(* Logix 5000 project; controller QW361 vendor 1 type 14 code 107 rev 32.11; software revision 32.00; part 12 of 20 *)

        [1618].time.Day := 29, [1618].time.Hour := 12, [1618].time.Minute := 24, [1618].time.Second := 59, [1618].time.DST_ON := 1, [1619].log_data[0].min := 1.0, [1619].log_data[0].max := 1.0, [1619].log_data[0].total := 300.0, [1619].log_data[0].time := 300.0, [1619].log_data[0].minminute := 25, [1619].log_data[0].maxminute := 25, [1619].log_data[0].valid := 1, [1619].log_data[1].valid := 1, [1619].log_data[2].valid := 1, [1619].log_data[3].valid := 1, [1619].log_data[4].valid := 1, [1619].time.Year := 2022, [1619].time.Month := 4, [1619].time.Day := 29, [1619].time.Hour := 12, [1619].time.Minute := 29, [1619].time.Second := 59, [1619].time.DST_ON := 1, [1620].log_data[0].min := 1.0, [1620].log_data[0].max := 1.0, [1620].log_data[0].total := 300.0, [1620].log_data[0].time := 300.0, [1620].log_data[0].minminute := 30, [1620].log_data[0].maxminute := 30, [1620].log_data[0].valid := 1, [1620].log_data[1].valid := 1, [1620].log_data[2].valid := 1, [1620].log_data[3].valid := 1, [1620].log_data[4].valid := 1, [1620].time.Year := 2022, [1620].time.Month := 4, [1620].time.Day := 29, [1620].time.Hour := 12, [1620].time.Minute := 34, [1620].time.Second := 59, [1620].time.DST_ON := 1, [1621].log_data[0].min := 1.0, [1621].log_data[0].max := 1.0, [1621].log_data[0].total := 300.0, [1621].log_data[0].time := 300.0, [1621].log_data[0].minminute := 35, [1621].log_data[0].maxminute := 35, [1621].log_data[0].valid := 1, [1621].log_data[1].valid := 1, [1621].log_data[2].valid := 1, [1621].log_data[3].valid := 1, [1621].log_data[4].valid := 1, [1621].time.Year := 2022, [1621].time.Month := 4, [1621].time.Day := 29, [1621].time.Hour := 12, [1621].time.Minute := 39, [1621].time.Second := 59, [1621].time.DST_ON := 1, [1622].log_data[0].min := 1.0,
        [1622].log_data[0].max := 1.0, [1622].log_data[0].total := 300.0, [1622].log_data[0].time := 300.0, [1622].log_data[0].minminute := 40, [1622].log_data[0].maxminute := 40, [1622].log_data[0].valid := 1, [1622].log_data[1].valid := 1, [1622].log_data[2].valid := 1, [1622].log_data[3].valid := 1, [1622].log_data[4].valid := 1, [1622].time.Year := 2022, [1622].time.Month := 4, [1622].time.Day := 29, [1622].time.Hour := 12, [1622].time.Minute := 44, [1622].time.Second := 59, [1622].time.DST_ON := 1, [1623].log_data[0].min := 1.0, [1623].log_data[0].max := 1.0, [1623].log_data[0].total := 300.0, [1623].log_data[0].time := 300.0, [1623].log_data[0].minminute := 45, [1623].log_data[0].maxminute := 45, [1623].log_data[0].valid := 1, [1623].log_data[1].valid := 1, [1623].log_data[2].valid := 1, [1623].log_data[3].valid := 1, [1623].log_data[4].valid := 1, [1623].time.Year := 2022, [1623].time.Month := 4, [1623].time.Day := 29, [1623].time.Hour := 12, [1623].time.Minute := 49, [1623].time.Second := 59, [1623].time.DST_ON := 1, [1624].log_data[0].min := 1.0, [1624].log_data[0].max := 1.0, [1624].log_data[0].total := 300.0, [1624].log_data[0].time := 300.0, [1624].log_data[0].minminute := 50, [1624].log_data[0].maxminute := 50, [1624].log_data[0].valid := 1, [1624].log_data[1].valid := 1, [1624].log_data[2].valid := 1, [1624].log_data[3].valid := 1, [1624].log_data[4].valid := 1, [1624].time.Year := 2022, [1624].time.Month := 4, [1624].time.Day := 29, [1624].time.Hour := 12, [1624].time.Minute := 54, [1624].time.Second := 59, [1624].time.DST_ON := 1, [1625].log_data[0].min := 1.0, [1625].log_data[0].max := 1.0, [1625].log_data[0].total := 300.0, [1625].log_data[0].time := 300.0, [1625].log_data[0].minminute := 55, [1625].log_data[0].maxminute := 55, [1625].log_data[0].valid := 1,
        [1625].log_data[1].valid := 1, [1625].log_data[2].valid := 1, [1625].log_data[3].valid := 1, [1625].log_data[4].valid := 1, [1625].time.Year := 2022, [1625].time.Month := 4, [1625].time.Day := 29, [1625].time.Hour := 12, [1625].time.Minute := 59, [1625].time.Second := 59, [1625].time.DST_ON := 1, [1626].log_data[0].min := 1.0, [1626].log_data[0].max := 1.0, [1626].log_data[0].total := 300.0, [1626].log_data[0].time := 300.0, [1626].log_data[0].valid := 1, [1626].log_data[1].valid := 1, [1626].log_data[2].valid := 1, [1626].log_data[3].valid := 1, [1626].log_data[4].valid := 1, [1626].time.Year := 2022, [1626].time.Month := 4, [1626].time.Day := 29, [1626].time.Hour := 13, [1626].time.Minute := 4, [1626].time.Second := 59, [1626].time.DST_ON := 1, [1627].log_data[0].min := 1.0, [1627].log_data[0].max := 1.0, [1627].log_data[0].total := 300.0, [1627].log_data[0].time := 300.0, [1627].log_data[0].minminute := 5, [1627].log_data[0].maxminute := 5, [1627].log_data[0].valid := 1, [1627].log_data[1].valid := 1, [1627].log_data[2].valid := 1, [1627].log_data[3].valid := 1, [1627].log_data[4].valid := 1, [1627].time.Year := 2022, [1627].time.Month := 4, [1627].time.Day := 29, [1627].time.Hour := 13, [1627].time.Minute := 9, [1627].time.Second := 59, [1627].time.DST_ON := 1, [1628].log_data[0].min := 1.0, [1628].log_data[0].max := 1.0, [1628].log_data[0].total := 300.0, [1628].log_data[0].time := 300.0, [1628].log_data[0].minminute := 10, [1628].log_data[0].maxminute := 10, [1628].log_data[0].valid := 1, [1628].log_data[1].valid := 1, [1628].log_data[2].valid := 1, [1628].log_data[3].valid := 1, [1628].log_data[4].valid := 1, [1628].time.Year := 2022, [1628].time.Month := 4, [1628].time.Day := 29, [1628].time.Hour := 13,
        [1628].time.Minute := 14, [1628].time.Second := 59, [1628].time.DST_ON := 1, [1629].log_data[0].min := 1.0, [1629].log_data[0].max := 1.0, [1629].log_data[0].total := 300.0, [1629].log_data[0].time := 300.0, [1629].log_data[0].minminute := 15, [1629].log_data[0].maxminute := 15, [1629].log_data[0].valid := 1, [1629].log_data[1].valid := 1, [1629].log_data[2].valid := 1, [1629].log_data[3].valid := 1, [1629].log_data[4].valid := 1, [1629].time.Year := 2022, [1629].time.Month := 4, [1629].time.Day := 29, [1629].time.Hour := 13, [1629].time.Minute := 19, [1629].time.Second := 59, [1629].time.DST_ON := 1, [1630].log_data[0].min := 1.0, [1630].log_data[0].max := 1.0, [1630].log_data[0].total := 300.0, [1630].log_data[0].time := 300.0, [1630].log_data[0].minminute := 20, [1630].log_data[0].maxminute := 20, [1630].log_data[0].valid := 1, [1630].log_data[1].valid := 1, [1630].log_data[2].valid := 1, [1630].log_data[3].valid := 1, [1630].log_data[4].valid := 1, [1630].time.Year := 2022, [1630].time.Month := 4, [1630].time.Day := 29, [1630].time.Hour := 13, [1630].time.Minute := 24, [1630].time.Second := 59, [1630].time.DST_ON := 1, [1631].log_data[0].min := 1.0, [1631].log_data[0].max := 1.0, [1631].log_data[0].total := 300.0, [1631].log_data[0].time := 300.0, [1631].log_data[0].minminute := 25, [1631].log_data[0].maxminute := 25, [1631].log_data[0].valid := 1, [1631].log_data[1].valid := 1, [1631].log_data[2].valid := 1, [1631].log_data[3].valid := 1, [1631].log_data[4].valid := 1, [1631].time.Year := 2022, [1631].time.Month := 4, [1631].time.Day := 29, [1631].time.Hour := 13, [1631].time.Minute := 29, [1631].time.Second := 59, [1631].time.DST_ON := 1, [1632].log_data[0].min := 1.0, [1632].log_data[0].max := 1.0, [1632].log_data[0].total := 300.0,
        [1632].log_data[0].time := 300.0, [1632].log_data[0].minminute := 30, [1632].log_data[0].maxminute := 30, [1632].log_data[0].valid := 1, [1632].log_data[1].valid := 1, [1632].log_data[2].valid := 1, [1632].log_data[3].valid := 1, [1632].log_data[4].valid := 1, [1632].time.Year := 2022, [1632].time.Month := 4, [1632].time.Day := 29, [1632].time.Hour := 13, [1632].time.Minute := 34, [1632].time.Second := 59, [1632].time.DST_ON := 1, [1633].log_data[0].min := 1.0, [1633].log_data[0].max := 1.0, [1633].log_data[0].total := 300.001, [1633].log_data[0].time := 300.001, [1633].log_data[0].minminute := 35, [1633].log_data[0].maxminute := 35, [1633].log_data[0].valid := 1, [1633].log_data[1].valid := 1, [1633].log_data[2].valid := 1, [1633].log_data[3].valid := 1, [1633].log_data[4].valid := 1, [1633].time.Year := 2022, [1633].time.Month := 4, [1633].time.Day := 29, [1633].time.Hour := 13, [1633].time.Minute := 39, [1633].time.Second := 59, [1633].time.DST_ON := 1, [1634].log_data[0].min := 1.0, [1634].log_data[0].max := 1.0, [1634].log_data[0].total := 300.0, [1634].log_data[0].time := 300.0, [1634].log_data[0].minminute := 40, [1634].log_data[0].maxminute := 40, [1634].log_data[0].valid := 1, [1634].log_data[1].valid := 1, [1634].log_data[2].valid := 1, [1634].log_data[3].valid := 1, [1634].log_data[4].valid := 1, [1634].time.Year := 2022, [1634].time.Month := 4, [1634].time.Day := 29, [1634].time.Hour := 13, [1634].time.Minute := 44, [1634].time.Second := 59, [1634].time.DST_ON := 1, [1635].log_data[0].min := 1.0, [1635].log_data[0].max := 1.0, [1635].log_data[0].total := 300.0, [1635].log_data[0].time := 300.0, [1635].log_data[0].minminute := 45, [1635].log_data[0].maxminute := 45, [1635].log_data[0].valid := 1, [1635].log_data[1].valid := 1, [1635].log_data[2].valid := 1,
        [1635].log_data[3].valid := 1, [1635].log_data[4].valid := 1, [1635].time.Year := 2022, [1635].time.Month := 4, [1635].time.Day := 29, [1635].time.Hour := 13, [1635].time.Minute := 49, [1635].time.Second := 59, [1635].time.DST_ON := 1, [1636].log_data[0].min := 1.0, [1636].log_data[0].max := 1.0, [1636].log_data[0].total := 300.0, [1636].log_data[0].time := 300.0, [1636].log_data[0].minminute := 50, [1636].log_data[0].maxminute := 50, [1636].log_data[0].valid := 1, [1636].log_data[1].valid := 1, [1636].log_data[2].valid := 1, [1636].log_data[3].valid := 1, [1636].log_data[4].valid := 1, [1636].time.Year := 2022, [1636].time.Month := 4, [1636].time.Day := 29, [1636].time.Hour := 13, [1636].time.Minute := 54, [1636].time.Second := 59, [1636].time.DST_ON := 1, [1637].log_data[0].min := 1.0, [1637].log_data[0].max := 1.0, [1637].log_data[0].total := 300.0, [1637].log_data[0].time := 300.0, [1637].log_data[0].minminute := 55, [1637].log_data[0].maxminute := 55, [1637].log_data[0].valid := 1, [1637].log_data[1].valid := 1, [1637].log_data[2].valid := 1, [1637].log_data[3].valid := 1, [1637].log_data[4].valid := 1, [1637].time.Year := 2022, [1637].time.Month := 4, [1637].time.Day := 29, [1637].time.Hour := 13, [1637].time.Minute := 59, [1637].time.Second := 59, [1637].time.DST_ON := 1, [1638].log_data[0].min := 1.0, [1638].log_data[0].max := 1.0, [1638].log_data[0].total := 300.0, [1638].log_data[0].time := 300.0, [1638].log_data[0].valid := 1, [1638].log_data[1].valid := 1, [1638].log_data[2].valid := 1, [1638].log_data[3].valid := 1, [1638].log_data[4].valid := 1, [1638].time.Year := 2022, [1638].time.Month := 4, [1638].time.Day := 29, [1638].time.Hour := 14, [1638].time.Minute := 4, [1638].time.Second := 59,
        [1638].time.DST_ON := 1, [1639].log_data[0].min := 1.0, [1639].log_data[0].max := 1.0, [1639].log_data[0].total := 300.0, [1639].log_data[0].time := 300.0, [1639].log_data[0].minminute := 5, [1639].log_data[0].maxminute := 5, [1639].log_data[0].valid := 1, [1639].log_data[1].valid := 1, [1639].log_data[2].valid := 1, [1639].log_data[3].valid := 1, [1639].log_data[4].valid := 1, [1639].time.Year := 2022, [1639].time.Month := 4, [1639].time.Day := 29, [1639].time.Hour := 14, [1639].time.Minute := 9, [1639].time.Second := 59, [1639].time.DST_ON := 1, [1640].log_data[0].min := 1.0, [1640].log_data[0].max := 1.0, [1640].log_data[0].total := 300.0, [1640].log_data[0].time := 300.0, [1640].log_data[0].minminute := 10, [1640].log_data[0].maxminute := 10, [1640].log_data[0].valid := 1, [1640].log_data[1].valid := 1, [1640].log_data[2].valid := 1, [1640].log_data[3].valid := 1, [1640].log_data[4].valid := 1, [1640].time.Year := 2022, [1640].time.Month := 4, [1640].time.Day := 29, [1640].time.Hour := 14, [1640].time.Minute := 14, [1640].time.Second := 59, [1640].time.DST_ON := 1, [1641].log_data[0].min := 1.0, [1641].log_data[0].max := 1.0, [1641].log_data[0].total := 299.999, [1641].log_data[0].time := 299.999, [1641].log_data[0].minminute := 15, [1641].log_data[0].maxminute := 15, [1641].log_data[0].valid := 1, [1641].log_data[1].valid := 1, [1641].log_data[2].valid := 1, [1641].log_data[3].valid := 1, [1641].log_data[4].valid := 1, [1641].time.Year := 2022, [1641].time.Month := 4, [1641].time.Day := 29, [1641].time.Hour := 14, [1641].time.Minute := 19, [1641].time.Second := 59, [1641].time.DST_ON := 1, [1642].log_data[0].min := 1.0, [1642].log_data[0].max := 1.0, [1642].log_data[0].total := 300.0, [1642].log_data[0].time := 300.0, [1642].log_data[0].minminute := 20,
        [1642].log_data[0].maxminute := 20, [1642].log_data[0].valid := 1, [1642].log_data[1].valid := 1, [1642].log_data[2].valid := 1, [1642].log_data[3].valid := 1, [1642].log_data[4].valid := 1, [1642].time.Year := 2022, [1642].time.Month := 4, [1642].time.Day := 29, [1642].time.Hour := 14, [1642].time.Minute := 24, [1642].time.Second := 59, [1642].time.DST_ON := 1, [1643].log_data[0].min := 1.0, [1643].log_data[0].max := 1.0, [1643].log_data[0].total := 300.0, [1643].log_data[0].time := 300.0, [1643].log_data[0].minminute := 25, [1643].log_data[0].maxminute := 25, [1643].log_data[0].valid := 1, [1643].log_data[1].valid := 1, [1643].log_data[2].valid := 1, [1643].log_data[3].valid := 1, [1643].log_data[4].valid := 1, [1643].time.Year := 2022, [1643].time.Month := 4, [1643].time.Day := 29, [1643].time.Hour := 14, [1643].time.Minute := 29, [1643].time.Second := 59, [1643].time.DST_ON := 1, [1644].log_data[0].min := 1.0, [1644].log_data[0].max := 1.0, [1644].log_data[0].total := 300.0, [1644].log_data[0].time := 300.0, [1644].log_data[0].minminute := 30, [1644].log_data[0].maxminute := 30, [1644].log_data[0].valid := 1, [1644].log_data[1].valid := 1, [1644].log_data[2].valid := 1, [1644].log_data[3].valid := 1, [1644].log_data[4].valid := 1, [1644].time.Year := 2022, [1644].time.Month := 4, [1644].time.Day := 29, [1644].time.Hour := 14, [1644].time.Minute := 34, [1644].time.Second := 59, [1644].time.DST_ON := 1, [1645].log_data[0].min := 1.0, [1645].log_data[0].max := 1.0, [1645].log_data[0].total := 300.0, [1645].log_data[0].time := 300.0, [1645].log_data[0].minminute := 35, [1645].log_data[0].maxminute := 35, [1645].log_data[0].valid := 1, [1645].log_data[1].valid := 1, [1645].log_data[2].valid := 1, [1645].log_data[3].valid := 1, [1645].log_data[4].valid := 1,
        [1645].time.Year := 2022, [1645].time.Month := 4, [1645].time.Day := 29, [1645].time.Hour := 14, [1645].time.Minute := 39, [1645].time.Second := 59, [1645].time.DST_ON := 1, [1646].log_data[0].min := 1.0, [1646].log_data[0].max := 1.0, [1646].log_data[0].total := 300.0, [1646].log_data[0].time := 300.0, [1646].log_data[0].minminute := 40, [1646].log_data[0].maxminute := 40, [1646].log_data[0].valid := 1, [1646].log_data[1].valid := 1, [1646].log_data[2].valid := 1, [1646].log_data[3].valid := 1, [1646].log_data[4].valid := 1, [1646].time.Year := 2022, [1646].time.Month := 4, [1646].time.Day := 29, [1646].time.Hour := 14, [1646].time.Minute := 44, [1646].time.Second := 59, [1646].time.DST_ON := 1, [1647].log_data[0].min := 1.0, [1647].log_data[0].max := 1.0, [1647].log_data[0].total := 300.0, [1647].log_data[0].time := 300.0, [1647].log_data[0].minminute := 45, [1647].log_data[0].maxminute := 45, [1647].log_data[0].valid := 1, [1647].log_data[1].valid := 1, [1647].log_data[2].valid := 1, [1647].log_data[3].valid := 1, [1647].log_data[4].valid := 1, [1647].time.Year := 2022, [1647].time.Month := 4, [1647].time.Day := 29, [1647].time.Hour := 14, [1647].time.Minute := 49, [1647].time.Second := 59, [1647].time.DST_ON := 1, [1648].log_data[0].min := 1.0, [1648].log_data[0].max := 1.0, [1648].log_data[0].total := 300.0, [1648].log_data[0].time := 300.0, [1648].log_data[0].minminute := 50, [1648].log_data[0].maxminute := 50, [1648].log_data[0].valid := 1, [1648].log_data[1].valid := 1, [1648].log_data[2].valid := 1, [1648].log_data[3].valid := 1, [1648].log_data[4].valid := 1, [1648].time.Year := 2022, [1648].time.Month := 4, [1648].time.Day := 29, [1648].time.Hour := 14, [1648].time.Minute := 54, [1648].time.Second := 59,
        [1648].time.DST_ON := 1, [1649].log_data[0].min := 1.0, [1649].log_data[0].max := 1.0, [1649].log_data[0].total := 300.0, [1649].log_data[0].time := 300.0, [1649].log_data[0].minminute := 55, [1649].log_data[0].maxminute := 55, [1649].log_data[0].valid := 1, [1649].log_data[1].valid := 1, [1649].log_data[2].valid := 1, [1649].log_data[3].valid := 1, [1649].log_data[4].valid := 1, [1649].time.Year := 2022, [1649].time.Month := 4, [1649].time.Day := 29, [1649].time.Hour := 14, [1649].time.Minute := 59, [1649].time.Second := 59, [1649].time.DST_ON := 1, [1650].log_data[0].min := 1.0, [1650].log_data[0].max := 1.0, [1650].log_data[0].total := 300.0, [1650].log_data[0].time := 300.0, [1650].log_data[0].valid := 1, [1650].log_data[1].valid := 1, [1650].log_data[2].valid := 1, [1650].log_data[3].valid := 1, [1650].log_data[4].valid := 1, [1650].time.Year := 2022, [1650].time.Month := 4, [1650].time.Day := 29, [1650].time.Hour := 15, [1650].time.Minute := 4, [1650].time.Second := 59, [1650].time.DST_ON := 1, [1651].log_data[0].min := 1.0, [1651].log_data[0].max := 1.0, [1651].log_data[0].total := 300.0, [1651].log_data[0].time := 300.0, [1651].log_data[0].minminute := 5, [1651].log_data[0].maxminute := 5, [1651].log_data[0].valid := 1, [1651].log_data[1].valid := 1, [1651].log_data[2].valid := 1, [1651].log_data[3].valid := 1, [1651].log_data[4].valid := 1, [1651].time.Year := 2022, [1651].time.Month := 4, [1651].time.Day := 29, [1651].time.Hour := 15, [1651].time.Minute := 9, [1651].time.Second := 59, [1651].time.DST_ON := 1, [1652].log_data[0].min := 1.0, [1652].log_data[0].max := 1.0, [1652].log_data[0].total := 300.0, [1652].log_data[0].time := 300.0, [1652].log_data[0].minminute := 10, [1652].log_data[0].maxminute := 10, [1652].log_data[0].valid := 1,
        [1652].log_data[1].valid := 1, [1652].log_data[2].valid := 1, [1652].log_data[3].valid := 1, [1652].log_data[4].valid := 1, [1652].time.Year := 2022, [1652].time.Month := 4, [1652].time.Day := 29, [1652].time.Hour := 15, [1652].time.Minute := 14, [1652].time.Second := 59, [1652].time.DST_ON := 1, [1653].log_data[0].min := 1.0, [1653].log_data[0].max := 1.0, [1653].log_data[0].total := 300.0, [1653].log_data[0].time := 300.0, [1653].log_data[0].minminute := 15, [1653].log_data[0].maxminute := 15, [1653].log_data[0].valid := 1, [1653].log_data[1].valid := 1, [1653].log_data[2].valid := 1, [1653].log_data[3].valid := 1, [1653].log_data[4].valid := 1, [1653].time.Year := 2022, [1653].time.Month := 4, [1653].time.Day := 29, [1653].time.Hour := 15, [1653].time.Minute := 19, [1653].time.Second := 59, [1653].time.DST_ON := 1, [1654].log_data[0].min := 1.0, [1654].log_data[0].max := 1.0, [1654].log_data[0].total := 300.0, [1654].log_data[0].time := 300.0, [1654].log_data[0].minminute := 20, [1654].log_data[0].maxminute := 20, [1654].log_data[0].valid := 1, [1654].log_data[1].valid := 1, [1654].log_data[2].valid := 1, [1654].log_data[3].valid := 1, [1654].log_data[4].valid := 1, [1654].time.Year := 2022, [1654].time.Month := 4, [1654].time.Day := 29, [1654].time.Hour := 15, [1654].time.Minute := 24, [1654].time.Second := 59, [1654].time.DST_ON := 1, [1655].log_data[0].min := 1.0, [1655].log_data[0].max := 1.0, [1655].log_data[0].total := 300.0, [1655].log_data[0].time := 300.0, [1655].log_data[0].minminute := 25, [1655].log_data[0].maxminute := 25, [1655].log_data[0].valid := 1, [1655].log_data[1].valid := 1, [1655].log_data[2].valid := 1, [1655].log_data[3].valid := 1, [1655].log_data[4].valid := 1, [1655].time.Year := 2022, [1655].time.Month := 4,
        [1655].time.Day := 29, [1655].time.Hour := 15, [1655].time.Minute := 29, [1655].time.Second := 59, [1655].time.DST_ON := 1, [1656].log_data[0].min := 1.0, [1656].log_data[0].max := 1.0, [1656].log_data[0].total := 300.001, [1656].log_data[0].time := 300.001, [1656].log_data[0].minminute := 30, [1656].log_data[0].maxminute := 30, [1656].log_data[0].valid := 1, [1656].log_data[1].valid := 1, [1656].log_data[2].valid := 1, [1656].log_data[3].valid := 1, [1656].log_data[4].valid := 1, [1656].time.Year := 2022, [1656].time.Month := 4, [1656].time.Day := 29, [1656].time.Hour := 15, [1656].time.Minute := 34, [1656].time.Second := 59, [1656].time.DST_ON := 1, [1657].log_data[0].min := 1.0, [1657].log_data[0].max := 1.0, [1657].log_data[0].total := 300.0, [1657].log_data[0].time := 300.0, [1657].log_data[0].minminute := 35, [1657].log_data[0].maxminute := 35, [1657].log_data[0].valid := 1, [1657].log_data[1].valid := 1, [1657].log_data[2].valid := 1, [1657].log_data[3].valid := 1, [1657].log_data[4].valid := 1, [1657].time.Year := 2022, [1657].time.Month := 4, [1657].time.Day := 29, [1657].time.Hour := 15, [1657].time.Minute := 39, [1657].time.Second := 59, [1657].time.DST_ON := 1, [1658].log_data[0].min := 1.0, [1658].log_data[0].max := 1.0, [1658].log_data[0].total := 300.0, [1658].log_data[0].time := 300.0, [1658].log_data[0].minminute := 40, [1658].log_data[0].maxminute := 40, [1658].log_data[0].valid := 1, [1658].log_data[1].valid := 1, [1658].log_data[2].valid := 1, [1658].log_data[3].valid := 1, [1658].log_data[4].valid := 1, [1658].time.Year := 2022, [1658].time.Month := 4, [1658].time.Day := 29, [1658].time.Hour := 15, [1658].time.Minute := 44, [1658].time.Second := 59, [1658].time.DST_ON := 1, [1659].log_data[0].min := 1.0,
        [1659].log_data[0].max := 1.0, [1659].log_data[0].total := 300.0, [1659].log_data[0].time := 300.0, [1659].log_data[0].minminute := 45, [1659].log_data[0].maxminute := 45, [1659].log_data[0].valid := 1, [1659].log_data[1].valid := 1, [1659].log_data[2].valid := 1, [1659].log_data[3].valid := 1, [1659].log_data[4].valid := 1, [1659].time.Year := 2022, [1659].time.Month := 4, [1659].time.Day := 29, [1659].time.Hour := 15, [1659].time.Minute := 49, [1659].time.Second := 59, [1659].time.DST_ON := 1, [1660].log_data[0].min := 1.0, [1660].log_data[0].max := 1.0, [1660].log_data[0].total := 300.0, [1660].log_data[0].time := 300.0, [1660].log_data[0].minminute := 50, [1660].log_data[0].maxminute := 50, [1660].log_data[0].valid := 1, [1660].log_data[1].valid := 1, [1660].log_data[2].valid := 1, [1660].log_data[3].valid := 1, [1660].log_data[4].valid := 1, [1660].time.Year := 2022, [1660].time.Month := 4, [1660].time.Day := 29, [1660].time.Hour := 15, [1660].time.Minute := 54, [1660].time.Second := 59, [1660].time.DST_ON := 1, [1661].log_data[0].min := 1.0, [1661].log_data[0].max := 1.0, [1661].log_data[0].total := 300.0, [1661].log_data[0].time := 300.0, [1661].log_data[0].minminute := 55, [1661].log_data[0].maxminute := 55, [1661].log_data[0].valid := 1, [1661].log_data[1].valid := 1, [1661].log_data[2].valid := 1, [1661].log_data[3].valid := 1, [1661].log_data[4].valid := 1, [1661].time.Year := 2022, [1661].time.Month := 4, [1661].time.Day := 29, [1661].time.Hour := 15, [1661].time.Minute := 59, [1661].time.Second := 59, [1661].time.DST_ON := 1, [1662].log_data[0].min := 1.0, [1662].log_data[0].max := 1.0, [1662].log_data[0].total := 300.0, [1662].log_data[0].time := 300.0, [1662].log_data[0].valid := 1, [1662].log_data[1].valid := 1, [1662].log_data[2].valid := 1,
        [1662].log_data[3].valid := 1, [1662].log_data[4].valid := 1, [1662].time.Year := 2022, [1662].time.Month := 4, [1662].time.Day := 29, [1662].time.Hour := 16, [1662].time.Minute := 4, [1662].time.Second := 59, [1662].time.DST_ON := 1, [1663].log_data[0].min := 1.0, [1663].log_data[0].max := 1.0, [1663].log_data[0].total := 300.0, [1663].log_data[0].time := 300.0, [1663].log_data[0].minminute := 5, [1663].log_data[0].maxminute := 5, [1663].log_data[0].valid := 1, [1663].log_data[1].valid := 1, [1663].log_data[2].valid := 1, [1663].log_data[3].valid := 1, [1663].log_data[4].valid := 1, [1663].time.Year := 2022, [1663].time.Month := 4, [1663].time.Day := 29, [1663].time.Hour := 16, [1663].time.Minute := 9, [1663].time.Second := 59, [1663].time.DST_ON := 1, [1664].log_data[0].min := 1.0, [1664].log_data[0].max := 1.0, [1664].log_data[0].total := 300.0, [1664].log_data[0].time := 300.0, [1664].log_data[0].minminute := 10, [1664].log_data[0].maxminute := 10, [1664].log_data[0].valid := 1, [1664].log_data[1].valid := 1, [1664].log_data[2].valid := 1, [1664].log_data[3].valid := 1, [1664].log_data[4].valid := 1, [1664].time.Year := 2022, [1664].time.Month := 4, [1664].time.Day := 29, [1664].time.Hour := 16, [1664].time.Minute := 14, [1664].time.Second := 59, [1664].time.DST_ON := 1, [1665].log_data[0].min := 1.0, [1665].log_data[0].max := 1.0, [1665].log_data[0].total := 300.0, [1665].log_data[0].time := 300.0, [1665].log_data[0].minminute := 15, [1665].log_data[0].maxminute := 15, [1665].log_data[0].valid := 1, [1665].log_data[1].valid := 1, [1665].log_data[2].valid := 1, [1665].log_data[3].valid := 1, [1665].log_data[4].valid := 1, [1665].time.Year := 2022, [1665].time.Month := 4, [1665].time.Day := 29, [1665].time.Hour := 16,
        [1665].time.Minute := 19, [1665].time.Second := 59, [1665].time.DST_ON := 1, [1666].log_data[0].min := 1.0, [1666].log_data[0].max := 1.0, [1666].log_data[0].total := 300.0, [1666].log_data[0].time := 300.0, [1666].log_data[0].minminute := 20, [1666].log_data[0].maxminute := 20, [1666].log_data[0].valid := 1, [1666].log_data[1].valid := 1, [1666].log_data[2].valid := 1, [1666].log_data[3].valid := 1, [1666].log_data[4].valid := 1, [1666].time.Year := 2022, [1666].time.Month := 4, [1666].time.Day := 29, [1666].time.Hour := 16, [1666].time.Minute := 24, [1666].time.Second := 59, [1666].time.DST_ON := 1, [1667].log_data[0].min := 1.0, [1667].log_data[0].max := 1.0, [1667].log_data[0].total := 300.0, [1667].log_data[0].time := 300.0, [1667].log_data[0].minminute := 25, [1667].log_data[0].maxminute := 25, [1667].log_data[0].valid := 1, [1667].log_data[1].valid := 1, [1667].log_data[2].valid := 1, [1667].log_data[3].valid := 1, [1667].log_data[4].valid := 1, [1667].time.Year := 2022, [1667].time.Month := 4, [1667].time.Day := 29, [1667].time.Hour := 16, [1667].time.Minute := 29, [1667].time.Second := 59, [1667].time.DST_ON := 1, [1668].log_data[0].min := 1.0, [1668].log_data[0].max := 1.0, [1668].log_data[0].total := 300.0, [1668].log_data[0].time := 300.0, [1668].log_data[0].minminute := 30, [1668].log_data[0].maxminute := 30, [1668].log_data[0].valid := 1, [1668].log_data[1].valid := 1, [1668].log_data[2].valid := 1, [1668].log_data[3].valid := 1, [1668].log_data[4].valid := 1, [1668].time.Year := 2022, [1668].time.Month := 4, [1668].time.Day := 29, [1668].time.Hour := 16, [1668].time.Minute := 34, [1668].time.Second := 59, [1668].time.DST_ON := 1, [1669].log_data[0].min := 1.0, [1669].log_data[0].max := 1.0, [1669].log_data[0].total := 300.0,
        [1669].log_data[0].time := 300.0, [1669].log_data[0].minminute := 35, [1669].log_data[0].maxminute := 35, [1669].log_data[0].valid := 1, [1669].log_data[1].valid := 1, [1669].log_data[2].valid := 1, [1669].log_data[3].valid := 1, [1669].log_data[4].valid := 1, [1669].time.Year := 2022, [1669].time.Month := 4, [1669].time.Day := 29, [1669].time.Hour := 16, [1669].time.Minute := 39, [1669].time.Second := 59, [1669].time.DST_ON := 1, [1670].log_data[0].min := 1.0, [1670].log_data[0].max := 1.0, [1670].log_data[0].total := 300.0, [1670].log_data[0].time := 300.0, [1670].log_data[0].minminute := 40, [1670].log_data[0].maxminute := 40, [1670].log_data[0].valid := 1, [1670].log_data[1].valid := 1, [1670].log_data[2].valid := 1, [1670].log_data[3].valid := 1, [1670].log_data[4].valid := 1, [1670].time.Year := 2022, [1670].time.Month := 4, [1670].time.Day := 29, [1670].time.Hour := 16, [1670].time.Minute := 44, [1670].time.Second := 59, [1670].time.DST_ON := 1, [1671].log_data[0].min := 1.0, [1671].log_data[0].max := 1.0, [1671].log_data[0].total := 300.0, [1671].log_data[0].time := 300.0, [1671].log_data[0].minminute := 45, [1671].log_data[0].maxminute := 45, [1671].log_data[0].valid := 1, [1671].log_data[1].valid := 1, [1671].log_data[2].valid := 1, [1671].log_data[3].valid := 1, [1671].log_data[4].valid := 1, [1671].time.Year := 2022, [1671].time.Month := 4, [1671].time.Day := 29, [1671].time.Hour := 16, [1671].time.Minute := 49, [1671].time.Second := 59, [1671].time.DST_ON := 1, [1672].log_data[0].min := 1.0, [1672].log_data[0].max := 1.0, [1672].log_data[0].total := 300.0, [1672].log_data[0].time := 300.0, [1672].log_data[0].minminute := 50, [1672].log_data[0].maxminute := 50, [1672].log_data[0].valid := 1, [1672].log_data[1].valid := 1, [1672].log_data[2].valid := 1,
        [1672].log_data[3].valid := 1, [1672].log_data[4].valid := 1, [1672].time.Year := 2022, [1672].time.Month := 4, [1672].time.Day := 29, [1672].time.Hour := 16, [1672].time.Minute := 54, [1672].time.Second := 59, [1672].time.DST_ON := 1, [1673].log_data[0].min := 1.0, [1673].log_data[0].max := 1.0, [1673].log_data[0].total := 300.0, [1673].log_data[0].time := 300.0, [1673].log_data[0].minminute := 55, [1673].log_data[0].maxminute := 55, [1673].log_data[0].valid := 1, [1673].log_data[1].valid := 1, [1673].log_data[2].valid := 1, [1673].log_data[3].valid := 1, [1673].log_data[4].valid := 1, [1673].time.Year := 2022, [1673].time.Month := 4, [1673].time.Day := 29, [1673].time.Hour := 16, [1673].time.Minute := 59, [1673].time.Second := 59, [1673].time.DST_ON := 1, [1674].log_data[0].min := 1.0, [1674].log_data[0].max := 1.0, [1674].log_data[0].total := 300.0, [1674].log_data[0].time := 300.0, [1674].log_data[0].valid := 1, [1674].log_data[1].valid := 1, [1674].log_data[2].valid := 1, [1674].log_data[3].valid := 1, [1674].log_data[4].valid := 1, [1674].time.Year := 2022, [1674].time.Month := 4, [1674].time.Day := 29, [1674].time.Hour := 17, [1674].time.Minute := 4, [1674].time.Second := 59, [1674].time.DST_ON := 1, [1675].log_data[0].min := 1.0, [1675].log_data[0].max := 1.0, [1675].log_data[0].total := 300.0, [1675].log_data[0].time := 300.0, [1675].log_data[0].minminute := 5, [1675].log_data[0].maxminute := 5, [1675].log_data[0].valid := 1, [1675].log_data[1].valid := 1, [1675].log_data[2].valid := 1, [1675].log_data[3].valid := 1, [1675].log_data[4].valid := 1, [1675].time.Year := 2022, [1675].time.Month := 4, [1675].time.Day := 29, [1675].time.Hour := 17, [1675].time.Minute := 9, [1675].time.Second := 59,
        [1675].time.DST_ON := 1, [1676].log_data[0].min := 1.0, [1676].log_data[0].max := 1.0, [1676].log_data[0].total := 300.0, [1676].log_data[0].time := 300.0, [1676].log_data[0].minminute := 10, [1676].log_data[0].maxminute := 10, [1676].log_data[0].valid := 1, [1676].log_data[1].valid := 1, [1676].log_data[2].valid := 1, [1676].log_data[3].valid := 1, [1676].log_data[4].valid := 1, [1676].time.Year := 2022, [1676].time.Month := 4, [1676].time.Day := 29, [1676].time.Hour := 17, [1676].time.Minute := 14, [1676].time.Second := 59, [1676].time.DST_ON := 1, [1677].log_data[0].min := 1.0, [1677].log_data[0].max := 1.0, [1677].log_data[0].total := 300.0, [1677].log_data[0].time := 300.0, [1677].log_data[0].minminute := 15, [1677].log_data[0].maxminute := 15, [1677].log_data[0].valid := 1, [1677].log_data[1].valid := 1, [1677].log_data[2].valid := 1, [1677].log_data[3].valid := 1, [1677].log_data[4].valid := 1, [1677].time.Year := 2022, [1677].time.Month := 4, [1677].time.Day := 29, [1677].time.Hour := 17, [1677].time.Minute := 19, [1677].time.Second := 59, [1677].time.DST_ON := 1, [1678].log_data[0].min := 1.0, [1678].log_data[0].max := 1.0, [1678].log_data[0].total := 299.999, [1678].log_data[0].time := 299.999, [1678].log_data[0].minminute := 20, [1678].log_data[0].maxminute := 20, [1678].log_data[0].valid := 1, [1678].log_data[1].valid := 1, [1678].log_data[2].valid := 1, [1678].log_data[3].valid := 1, [1678].log_data[4].valid := 1, [1678].time.Year := 2022, [1678].time.Month := 4, [1678].time.Day := 29, [1678].time.Hour := 17, [1678].time.Minute := 24, [1678].time.Second := 59, [1678].time.DST_ON := 1, [1679].log_data[0].min := 1.0, [1679].log_data[0].max := 1.0, [1679].log_data[0].total := 300.0, [1679].log_data[0].time := 300.0, [1679].log_data[0].minminute := 25,
        [1679].log_data[0].maxminute := 25, [1679].log_data[0].valid := 1, [1679].log_data[1].valid := 1, [1679].log_data[2].valid := 1, [1679].log_data[3].valid := 1, [1679].log_data[4].valid := 1, [1679].time.Year := 2022, [1679].time.Month := 4, [1679].time.Day := 29, [1679].time.Hour := 17, [1679].time.Minute := 29, [1679].time.Second := 59, [1679].time.DST_ON := 1, [1680].log_data[0].min := 1.0, [1680].log_data[0].max := 1.0, [1680].log_data[0].total := 300.0, [1680].log_data[0].time := 300.0, [1680].log_data[0].minminute := 30, [1680].log_data[0].maxminute := 30, [1680].log_data[0].valid := 1, [1680].log_data[1].valid := 1, [1680].log_data[2].valid := 1, [1680].log_data[3].valid := 1, [1680].log_data[4].valid := 1, [1680].time.Year := 2022, [1680].time.Month := 4, [1680].time.Day := 29, [1680].time.Hour := 17, [1680].time.Minute := 34, [1680].time.Second := 59, [1680].time.DST_ON := 1, [1681].log_data[0].min := 1.0, [1681].log_data[0].max := 1.0, [1681].log_data[0].total := 300.0, [1681].log_data[0].time := 300.0, [1681].log_data[0].minminute := 35, [1681].log_data[0].maxminute := 35, [1681].log_data[0].valid := 1, [1681].log_data[1].valid := 1, [1681].log_data[2].valid := 1, [1681].log_data[3].valid := 1, [1681].log_data[4].valid := 1, [1681].time.Year := 2022, [1681].time.Month := 4, [1681].time.Day := 29, [1681].time.Hour := 17, [1681].time.Minute := 39, [1681].time.Second := 59, [1681].time.DST_ON := 1, [1682].log_data[0].min := 1.0, [1682].log_data[0].max := 1.0, [1682].log_data[0].total := 300.0, [1682].log_data[0].time := 300.0, [1682].log_data[0].minminute := 40, [1682].log_data[0].maxminute := 40, [1682].log_data[0].valid := 1, [1682].log_data[1].valid := 1, [1682].log_data[2].valid := 1, [1682].log_data[3].valid := 1, [1682].log_data[4].valid := 1,
        [1682].time.Year := 2022, [1682].time.Month := 4, [1682].time.Day := 29, [1682].time.Hour := 17, [1682].time.Minute := 44, [1682].time.Second := 59, [1682].time.DST_ON := 1, [1683].log_data[0].min := 1.0, [1683].log_data[0].max := 1.0, [1683].log_data[0].total := 300.0, [1683].log_data[0].time := 300.0, [1683].log_data[0].minminute := 45, [1683].log_data[0].maxminute := 45, [1683].log_data[0].valid := 1, [1683].log_data[1].valid := 1, [1683].log_data[2].valid := 1, [1683].log_data[3].valid := 1, [1683].log_data[4].valid := 1, [1683].time.Year := 2022, [1683].time.Month := 4, [1683].time.Day := 29, [1683].time.Hour := 17, [1683].time.Minute := 49, [1683].time.Second := 59, [1683].time.DST_ON := 1, [1684].log_data[0].min := 1.0, [1684].log_data[0].max := 1.0, [1684].log_data[0].total := 300.0, [1684].log_data[0].time := 300.0, [1684].log_data[0].minminute := 50, [1684].log_data[0].maxminute := 50, [1684].log_data[0].valid := 1, [1684].log_data[1].valid := 1, [1684].log_data[2].valid := 1, [1684].log_data[3].valid := 1, [1684].log_data[4].valid := 1, [1684].time.Year := 2022, [1684].time.Month := 4, [1684].time.Day := 29, [1684].time.Hour := 17, [1684].time.Minute := 54, [1684].time.Second := 59, [1684].time.DST_ON := 1, [1685].log_data[0].min := 1.0, [1685].log_data[0].max := 1.0, [1685].log_data[0].total := 300.0, [1685].log_data[0].time := 300.0, [1685].log_data[0].minminute := 55, [1685].log_data[0].maxminute := 55, [1685].log_data[0].valid := 1, [1685].log_data[1].valid := 1, [1685].log_data[2].valid := 1, [1685].log_data[3].valid := 1, [1685].log_data[4].valid := 1, [1685].time.Year := 2022, [1685].time.Month := 4, [1685].time.Day := 29, [1685].time.Hour := 17, [1685].time.Minute := 59, [1685].time.Second := 59,
        [1685].time.DST_ON := 1, [1686].log_data[0].min := 1.0, [1686].log_data[0].max := 1.0, [1686].log_data[0].total := 300.0, [1686].log_data[0].time := 300.0, [1686].log_data[0].valid := 1, [1686].log_data[1].valid := 1, [1686].log_data[2].valid := 1, [1686].log_data[3].valid := 1, [1686].log_data[4].valid := 1, [1686].time.Year := 2022, [1686].time.Month := 4, [1686].time.Day := 29, [1686].time.Hour := 18, [1686].time.Minute := 4, [1686].time.Second := 59, [1686].time.DST_ON := 1, [1687].log_data[0].min := 1.0, [1687].log_data[0].max := 1.0, [1687].log_data[0].total := 300.0, [1687].log_data[0].time := 300.0, [1687].log_data[0].minminute := 5, [1687].log_data[0].maxminute := 5, [1687].log_data[0].valid := 1, [1687].log_data[1].valid := 1, [1687].log_data[2].valid := 1, [1687].log_data[3].valid := 1, [1687].log_data[4].valid := 1, [1687].time.Year := 2022, [1687].time.Month := 4, [1687].time.Day := 29, [1687].time.Hour := 18, [1687].time.Minute := 9, [1687].time.Second := 59, [1687].time.DST_ON := 1, [1688].log_data[0].min := 1.0, [1688].log_data[0].max := 1.0, [1688].log_data[0].total := 300.0, [1688].log_data[0].time := 300.0, [1688].log_data[0].minminute := 10, [1688].log_data[0].maxminute := 10, [1688].log_data[0].valid := 1, [1688].log_data[1].valid := 1, [1688].log_data[2].valid := 1, [1688].log_data[3].valid := 1, [1688].log_data[4].valid := 1, [1688].time.Year := 2022, [1688].time.Month := 4, [1688].time.Day := 29, [1688].time.Hour := 18, [1688].time.Minute := 14, [1688].time.Second := 59, [1688].time.DST_ON := 1, [1689].log_data[0].min := 1.0, [1689].log_data[0].max := 1.0, [1689].log_data[0].total := 300.0, [1689].log_data[0].time := 300.0, [1689].log_data[0].minminute := 15, [1689].log_data[0].maxminute := 15, [1689].log_data[0].valid := 1,
        [1689].log_data[1].valid := 1, [1689].log_data[2].valid := 1, [1689].log_data[3].valid := 1, [1689].log_data[4].valid := 1, [1689].time.Year := 2022, [1689].time.Month := 4, [1689].time.Day := 29, [1689].time.Hour := 18, [1689].time.Minute := 19, [1689].time.Second := 59, [1689].time.DST_ON := 1, [1690].log_data[0].min := 1.0, [1690].log_data[0].max := 1.0, [1690].log_data[0].total := 300.0, [1690].log_data[0].time := 300.0, [1690].log_data[0].minminute := 20, [1690].log_data[0].maxminute := 20, [1690].log_data[0].valid := 1, [1690].log_data[1].valid := 1, [1690].log_data[2].valid := 1, [1690].log_data[3].valid := 1, [1690].log_data[4].valid := 1, [1690].time.Year := 2022, [1690].time.Month := 4, [1690].time.Day := 29, [1690].time.Hour := 18, [1690].time.Minute := 24, [1690].time.Second := 59, [1690].time.DST_ON := 1, [1691].log_data[0].min := 1.0, [1691].log_data[0].max := 1.0, [1691].log_data[0].total := 300.0, [1691].log_data[0].time := 300.0, [1691].log_data[0].minminute := 25, [1691].log_data[0].maxminute := 25, [1691].log_data[0].valid := 1, [1691].log_data[1].valid := 1, [1691].log_data[2].valid := 1, [1691].log_data[3].valid := 1, [1691].log_data[4].valid := 1, [1691].time.Year := 2022, [1691].time.Month := 4, [1691].time.Day := 29, [1691].time.Hour := 18, [1691].time.Minute := 29, [1691].time.Second := 59, [1691].time.DST_ON := 1, [1692].log_data[0].min := 1.0, [1692].log_data[0].max := 1.0, [1692].log_data[0].total := 300.0, [1692].log_data[0].time := 300.0, [1692].log_data[0].minminute := 30, [1692].log_data[0].maxminute := 30, [1692].log_data[0].valid := 1, [1692].log_data[1].valid := 1, [1692].log_data[2].valid := 1, [1692].log_data[3].valid := 1, [1692].log_data[4].valid := 1, [1692].time.Year := 2022, [1692].time.Month := 4,
        [1692].time.Day := 29, [1692].time.Hour := 18, [1692].time.Minute := 34, [1692].time.Second := 59, [1692].time.DST_ON := 1, [1693].log_data[0].min := 1.0, [1693].log_data[0].max := 1.0, [1693].log_data[0].total := 300.0, [1693].log_data[0].time := 300.0, [1693].log_data[0].minminute := 35, [1693].log_data[0].maxminute := 35, [1693].log_data[0].valid := 1, [1693].log_data[1].valid := 1, [1693].log_data[2].valid := 1, [1693].log_data[3].valid := 1, [1693].log_data[4].valid := 1, [1693].time.Year := 2022, [1693].time.Month := 4, [1693].time.Day := 29, [1693].time.Hour := 18, [1693].time.Minute := 39, [1693].time.Second := 59, [1693].time.DST_ON := 1, [1694].log_data[0].min := 1.0, [1694].log_data[0].max := 1.0, [1694].log_data[0].total := 300.0, [1694].log_data[0].time := 300.0, [1694].log_data[0].minminute := 40, [1694].log_data[0].maxminute := 40, [1694].log_data[0].valid := 1, [1694].log_data[1].valid := 1, [1694].log_data[2].valid := 1, [1694].log_data[3].valid := 1, [1694].log_data[4].valid := 1, [1694].time.Year := 2022, [1694].time.Month := 4, [1694].time.Day := 29, [1694].time.Hour := 18, [1694].time.Minute := 44, [1694].time.Second := 59, [1694].time.DST_ON := 1, [1695].log_data[0].min := 1.0, [1695].log_data[0].max := 1.0, [1695].log_data[0].total := 300.0, [1695].log_data[0].time := 300.0, [1695].log_data[0].minminute := 45, [1695].log_data[0].maxminute := 45, [1695].log_data[0].valid := 1, [1695].log_data[1].valid := 1, [1695].log_data[2].valid := 1, [1695].log_data[3].valid := 1, [1695].log_data[4].valid := 1, [1695].time.Year := 2022, [1695].time.Month := 4, [1695].time.Day := 29, [1695].time.Hour := 18, [1695].time.Minute := 49, [1695].time.Second := 59, [1695].time.DST_ON := 1, [1696].log_data[0].min := 1.0,
        [1696].log_data[0].max := 1.0, [1696].log_data[0].total := 300.0, [1696].log_data[0].time := 300.0, [1696].log_data[0].minminute := 50, [1696].log_data[0].maxminute := 50, [1696].log_data[0].valid := 1, [1696].log_data[1].valid := 1, [1696].log_data[2].valid := 1, [1696].log_data[3].valid := 1, [1696].log_data[4].valid := 1, [1696].time.Year := 2022, [1696].time.Month := 4, [1696].time.Day := 29, [1696].time.Hour := 18, [1696].time.Minute := 54, [1696].time.Second := 59, [1696].time.DST_ON := 1, [1697].log_data[0].min := 1.0, [1697].log_data[0].max := 1.0, [1697].log_data[0].total := 300.0, [1697].log_data[0].time := 300.0, [1697].log_data[0].minminute := 55, [1697].log_data[0].maxminute := 55, [1697].log_data[0].valid := 1, [1697].log_data[1].valid := 1, [1697].log_data[2].valid := 1, [1697].log_data[3].valid := 1, [1697].log_data[4].valid := 1, [1697].time.Year := 2022, [1697].time.Month := 4, [1697].time.Day := 29, [1697].time.Hour := 18, [1697].time.Minute := 59, [1697].time.Second := 59, [1697].time.DST_ON := 1, [1698].log_data[0].min := 1.0, [1698].log_data[0].max := 1.0, [1698].log_data[0].total := 300.0, [1698].log_data[0].time := 300.0, [1698].log_data[0].valid := 1, [1698].log_data[1].valid := 1, [1698].log_data[2].valid := 1, [1698].log_data[3].valid := 1, [1698].log_data[4].valid := 1, [1698].time.Year := 2022, [1698].time.Month := 4, [1698].time.Day := 29, [1698].time.Hour := 19, [1698].time.Minute := 4, [1698].time.Second := 59, [1698].time.DST_ON := 1, [1699].log_data[0].min := 1.0, [1699].log_data[0].max := 1.0, [1699].log_data[0].total := 300.0, [1699].log_data[0].time := 300.0, [1699].log_data[0].minminute := 5, [1699].log_data[0].maxminute := 5, [1699].log_data[0].valid := 1, [1699].log_data[1].valid := 1, [1699].log_data[2].valid := 1,
        [1699].log_data[3].valid := 1, [1699].log_data[4].valid := 1, [1699].time.Year := 2022, [1699].time.Month := 4, [1699].time.Day := 29, [1699].time.Hour := 19, [1699].time.Minute := 9, [1699].time.Second := 59, [1699].time.DST_ON := 1, [1700].log_data[0].min := 1.0, [1700].log_data[0].max := 1.0, [1700].log_data[0].total := 300.0, [1700].log_data[0].time := 300.0, [1700].log_data[0].minminute := 10, [1700].log_data[0].maxminute := 10, [1700].log_data[0].valid := 1, [1700].log_data[1].valid := 1, [1700].log_data[2].valid := 1, [1700].log_data[3].valid := 1, [1700].log_data[4].valid := 1, [1700].time.Year := 2022, [1700].time.Month := 4, [1700].time.Day := 29, [1700].time.Hour := 19, [1700].time.Minute := 14, [1700].time.Second := 59, [1700].time.DST_ON := 1, [1701].log_data[0].min := 1.0, [1701].log_data[0].max := 1.0, [1701].log_data[0].total := 300.0, [1701].log_data[0].time := 300.0, [1701].log_data[0].minminute := 15, [1701].log_data[0].maxminute := 15, [1701].log_data[0].valid := 1, [1701].log_data[1].valid := 1, [1701].log_data[2].valid := 1, [1701].log_data[3].valid := 1, [1701].log_data[4].valid := 1, [1701].time.Year := 2022, [1701].time.Month := 4, [1701].time.Day := 29, [1701].time.Hour := 19, [1701].time.Minute := 19, [1701].time.Second := 59, [1701].time.DST_ON := 1, [1702].log_data[0].min := 1.0, [1702].log_data[0].max := 1.0, [1702].log_data[0].total := 300.0, [1702].log_data[0].time := 300.0, [1702].log_data[0].minminute := 20, [1702].log_data[0].maxminute := 20, [1702].log_data[0].valid := 1, [1702].log_data[1].valid := 1, [1702].log_data[2].valid := 1, [1702].log_data[3].valid := 1, [1702].log_data[4].valid := 1, [1702].time.Year := 2022, [1702].time.Month := 4, [1702].time.Day := 29, [1702].time.Hour := 19,
        [1702].time.Minute := 24, [1702].time.Second := 59, [1702].time.DST_ON := 1, [1703].log_data[0].min := 1.0, [1703].log_data[0].max := 1.0, [1703].log_data[0].total := 300.0, [1703].log_data[0].time := 300.0, [1703].log_data[0].minminute := 25, [1703].log_data[0].maxminute := 25, [1703].log_data[0].valid := 1, [1703].log_data[1].valid := 1, [1703].log_data[2].valid := 1, [1703].log_data[3].valid := 1, [1703].log_data[4].valid := 1, [1703].time.Year := 2022, [1703].time.Month := 4, [1703].time.Day := 29, [1703].time.Hour := 19, [1703].time.Minute := 29, [1703].time.Second := 59, [1703].time.DST_ON := 1, [1704].log_data[0].min := 1.0, [1704].log_data[0].max := 1.0, [1704].log_data[0].total := 300.0, [1704].log_data[0].time := 300.0, [1704].log_data[0].minminute := 30, [1704].log_data[0].maxminute := 30, [1704].log_data[0].valid := 1, [1704].log_data[1].valid := 1, [1704].log_data[2].valid := 1, [1704].log_data[3].valid := 1, [1704].log_data[4].valid := 1, [1704].time.Year := 2022, [1704].time.Month := 4, [1704].time.Day := 29, [1704].time.Hour := 19, [1704].time.Minute := 34, [1704].time.Second := 59, [1704].time.DST_ON := 1, [1705].log_data[0].min := 1.0, [1705].log_data[0].max := 1.0, [1705].log_data[0].total := 300.0, [1705].log_data[0].time := 300.0, [1705].log_data[0].minminute := 35, [1705].log_data[0].maxminute := 35, [1705].log_data[0].valid := 1, [1705].log_data[1].valid := 1, [1705].log_data[2].valid := 1, [1705].log_data[3].valid := 1, [1705].log_data[4].valid := 1, [1705].time.Year := 2022, [1705].time.Month := 4, [1705].time.Day := 29, [1705].time.Hour := 19, [1705].time.Minute := 39, [1705].time.Second := 59, [1705].time.DST_ON := 1, [1706].log_data[0].min := 1.0, [1706].log_data[0].max := 1.0, [1706].log_data[0].total := 300.0,
        [1706].log_data[0].time := 300.0, [1706].log_data[0].minminute := 40, [1706].log_data[0].maxminute := 40, [1706].log_data[0].valid := 1, [1706].log_data[1].valid := 1, [1706].log_data[2].valid := 1, [1706].log_data[3].valid := 1, [1706].log_data[4].valid := 1, [1706].time.Year := 2022, [1706].time.Month := 4, [1706].time.Day := 29, [1706].time.Hour := 19, [1706].time.Minute := 44, [1706].time.Second := 59, [1706].time.DST_ON := 1, [1707].log_data[0].min := 1.0, [1707].log_data[0].max := 1.0, [1707].log_data[0].total := 300.0, [1707].log_data[0].time := 300.0, [1707].log_data[0].minminute := 45, [1707].log_data[0].maxminute := 45, [1707].log_data[0].valid := 1, [1707].log_data[1].valid := 1, [1707].log_data[2].valid := 1, [1707].log_data[3].valid := 1, [1707].log_data[4].valid := 1, [1707].time.Year := 2022, [1707].time.Month := 4, [1707].time.Day := 29, [1707].time.Hour := 19, [1707].time.Minute := 49, [1707].time.Second := 59, [1707].time.DST_ON := 1, [1708].log_data[0].min := 1.0, [1708].log_data[0].max := 1.0, [1708].log_data[0].total := 300.0, [1708].log_data[0].time := 300.0, [1708].log_data[0].minminute := 50, [1708].log_data[0].maxminute := 50, [1708].log_data[0].valid := 1, [1708].log_data[1].valid := 1, [1708].log_data[2].valid := 1, [1708].log_data[3].valid := 1, [1708].log_data[4].valid := 1, [1708].time.Year := 2022, [1708].time.Month := 4, [1708].time.Day := 29, [1708].time.Hour := 19, [1708].time.Minute := 54, [1708].time.Second := 59, [1708].time.DST_ON := 1, [1709].log_data[0].min := 1.0, [1709].log_data[0].max := 1.0, [1709].log_data[0].total := 300.0, [1709].log_data[0].time := 300.0, [1709].log_data[0].minminute := 55, [1709].log_data[0].maxminute := 55, [1709].log_data[0].valid := 1, [1709].log_data[1].valid := 1, [1709].log_data[2].valid := 1,
        [1709].log_data[3].valid := 1, [1709].log_data[4].valid := 1, [1709].time.Year := 2022, [1709].time.Month := 4, [1709].time.Day := 29, [1709].time.Hour := 19, [1709].time.Minute := 59, [1709].time.Second := 59, [1709].time.DST_ON := 1, [1710].log_data[0].min := 1.0, [1710].log_data[0].max := 1.0, [1710].log_data[0].total := 300.0, [1710].log_data[0].time := 300.0, [1710].log_data[0].valid := 1, [1710].log_data[1].valid := 1, [1710].log_data[2].valid := 1, [1710].log_data[3].valid := 1, [1710].log_data[4].valid := 1, [1710].time.Year := 2022, [1710].time.Month := 4, [1710].time.Day := 29, [1710].time.Hour := 20, [1710].time.Minute := 4, [1710].time.Second := 59, [1710].time.DST_ON := 1, [1711].log_data[0].min := 1.0, [1711].log_data[0].max := 1.0, [1711].log_data[0].total := 300.0, [1711].log_data[0].time := 300.0, [1711].log_data[0].minminute := 5, [1711].log_data[0].maxminute := 5, [1711].log_data[0].valid := 1, [1711].log_data[1].valid := 1, [1711].log_data[2].valid := 1, [1711].log_data[3].valid := 1, [1711].log_data[4].valid := 1, [1711].time.Year := 2022, [1711].time.Month := 4, [1711].time.Day := 29, [1711].time.Hour := 20, [1711].time.Minute := 9, [1711].time.Second := 59, [1711].time.DST_ON := 1, [1712].log_data[0].min := 1.0, [1712].log_data[0].max := 1.0, [1712].log_data[0].total := 299.999, [1712].log_data[0].time := 299.999, [1712].log_data[0].minminute := 10, [1712].log_data[0].maxminute := 10, [1712].log_data[0].valid := 1, [1712].log_data[1].valid := 1, [1712].log_data[2].valid := 1, [1712].log_data[3].valid := 1, [1712].log_data[4].valid := 1, [1712].time.Year := 2022, [1712].time.Month := 4, [1712].time.Day := 29, [1712].time.Hour := 20, [1712].time.Minute := 14, [1712].time.Second := 59,
        [1712].time.DST_ON := 1, [1713].log_data[0].min := 1.0, [1713].log_data[0].max := 1.0, [1713].log_data[0].total := 300.0, [1713].log_data[0].time := 300.0, [1713].log_data[0].minminute := 15, [1713].log_data[0].maxminute := 15, [1713].log_data[0].valid := 1, [1713].log_data[1].valid := 1, [1713].log_data[2].valid := 1, [1713].log_data[3].valid := 1, [1713].log_data[4].valid := 1, [1713].time.Year := 2022, [1713].time.Month := 4, [1713].time.Day := 29, [1713].time.Hour := 20, [1713].time.Minute := 19, [1713].time.Second := 59, [1713].time.DST_ON := 1, [1714].log_data[0].min := 1.0, [1714].log_data[0].max := 1.0, [1714].log_data[0].total := 300.0, [1714].log_data[0].time := 300.0, [1714].log_data[0].minminute := 20, [1714].log_data[0].maxminute := 20, [1714].log_data[0].valid := 1, [1714].log_data[1].valid := 1, [1714].log_data[2].valid := 1, [1714].log_data[3].valid := 1, [1714].log_data[4].valid := 1, [1714].time.Year := 2022, [1714].time.Month := 4, [1714].time.Day := 29, [1714].time.Hour := 20, [1714].time.Minute := 24, [1714].time.Second := 59, [1714].time.DST_ON := 1, [1715].log_data[0].min := 1.0, [1715].log_data[0].max := 1.0, [1715].log_data[0].total := 300.0, [1715].log_data[0].time := 300.0, [1715].log_data[0].minminute := 25, [1715].log_data[0].maxminute := 25, [1715].log_data[0].valid := 1, [1715].log_data[1].valid := 1, [1715].log_data[2].valid := 1, [1715].log_data[3].valid := 1, [1715].log_data[4].valid := 1, [1715].time.Year := 2022, [1715].time.Month := 4, [1715].time.Day := 29, [1715].time.Hour := 20, [1715].time.Minute := 29, [1715].time.Second := 59, [1715].time.DST_ON := 1, [1716].log_data[0].min := 1.0, [1716].log_data[0].max := 1.0, [1716].log_data[0].total := 300.0, [1716].log_data[0].time := 300.0, [1716].log_data[0].minminute := 30,
        [1716].log_data[0].maxminute := 30, [1716].log_data[0].valid := 1, [1716].log_data[1].valid := 1, [1716].log_data[2].valid := 1, [1716].log_data[3].valid := 1, [1716].log_data[4].valid := 1, [1716].time.Year := 2022, [1716].time.Month := 4, [1716].time.Day := 29, [1716].time.Hour := 20, [1716].time.Minute := 34, [1716].time.Second := 59, [1716].time.DST_ON := 1, [1717].log_data[0].min := 1.0, [1717].log_data[0].max := 1.0, [1717].log_data[0].total := 300.0, [1717].log_data[0].time := 300.0, [1717].log_data[0].minminute := 35, [1717].log_data[0].maxminute := 35, [1717].log_data[0].valid := 1, [1717].log_data[1].valid := 1, [1717].log_data[2].valid := 1, [1717].log_data[3].valid := 1, [1717].log_data[4].valid := 1, [1717].time.Year := 2022, [1717].time.Month := 4, [1717].time.Day := 29, [1717].time.Hour := 20, [1717].time.Minute := 39, [1717].time.Second := 59, [1717].time.DST_ON := 1, [1718].log_data[0].min := 1.0, [1718].log_data[0].max := 1.0, [1718].log_data[0].total := 300.0, [1718].log_data[0].time := 300.0, [1718].log_data[0].minminute := 40, [1718].log_data[0].maxminute := 40, [1718].log_data[0].valid := 1, [1718].log_data[1].valid := 1, [1718].log_data[2].valid := 1, [1718].log_data[3].valid := 1, [1718].log_data[4].valid := 1, [1718].time.Year := 2022, [1718].time.Month := 4, [1718].time.Day := 29, [1718].time.Hour := 20, [1718].time.Minute := 44, [1718].time.Second := 59, [1718].time.DST_ON := 1, [1719].log_data[0].min := 1.0, [1719].log_data[0].max := 1.0, [1719].log_data[0].total := 300.0, [1719].log_data[0].time := 300.0, [1719].log_data[0].minminute := 45, [1719].log_data[0].maxminute := 45, [1719].log_data[0].valid := 1, [1719].log_data[1].valid := 1, [1719].log_data[2].valid := 1, [1719].log_data[3].valid := 1, [1719].log_data[4].valid := 1,
        [1719].time.Year := 2022, [1719].time.Month := 4, [1719].time.Day := 29, [1719].time.Hour := 20, [1719].time.Minute := 49, [1719].time.Second := 59, [1719].time.DST_ON := 1, [1720].log_data[0].min := 1.0, [1720].log_data[0].max := 1.0, [1720].log_data[0].total := 300.0, [1720].log_data[0].time := 300.0, [1720].log_data[0].minminute := 50, [1720].log_data[0].maxminute := 50, [1720].log_data[0].valid := 1, [1720].log_data[1].valid := 1, [1720].log_data[2].valid := 1, [1720].log_data[3].valid := 1, [1720].log_data[4].valid := 1, [1720].time.Year := 2022, [1720].time.Month := 4, [1720].time.Day := 29, [1720].time.Hour := 20, [1720].time.Minute := 54, [1720].time.Second := 59, [1720].time.DST_ON := 1, [1721].log_data[0].min := 1.0, [1721].log_data[0].max := 1.0, [1721].log_data[0].total := 300.0, [1721].log_data[0].time := 300.0, [1721].log_data[0].minminute := 55, [1721].log_data[0].maxminute := 55, [1721].log_data[0].valid := 1, [1721].log_data[1].valid := 1, [1721].log_data[2].valid := 1, [1721].log_data[3].valid := 1, [1721].log_data[4].valid := 1, [1721].time.Year := 2022, [1721].time.Month := 4, [1721].time.Day := 29, [1721].time.Hour := 20, [1721].time.Minute := 59, [1721].time.Second := 59, [1721].time.DST_ON := 1, [1722].log_data[0].min := 1.0, [1722].log_data[0].max := 1.0, [1722].log_data[0].total := 300.0, [1722].log_data[0].time := 300.0, [1722].log_data[0].valid := 1, [1722].log_data[1].valid := 1, [1722].log_data[2].valid := 1, [1722].log_data[3].valid := 1, [1722].log_data[4].valid := 1, [1722].time.Year := 2022, [1722].time.Month := 4, [1722].time.Day := 29, [1722].time.Hour := 21, [1722].time.Minute := 4, [1722].time.Second := 59, [1722].time.DST_ON := 1, [1723].log_data[0].min := 1.0,
        [1723].log_data[0].max := 1.0, [1723].log_data[0].total := 300.0, [1723].log_data[0].time := 300.0, [1723].log_data[0].minminute := 5, [1723].log_data[0].maxminute := 5, [1723].log_data[0].valid := 1, [1723].log_data[1].valid := 1, [1723].log_data[2].valid := 1, [1723].log_data[3].valid := 1, [1723].log_data[4].valid := 1, [1723].time.Year := 2022, [1723].time.Month := 4, [1723].time.Day := 29, [1723].time.Hour := 21, [1723].time.Minute := 9, [1723].time.Second := 59, [1723].time.DST_ON := 1, [1724].log_data[0].min := 1.0, [1724].log_data[0].max := 1.0, [1724].log_data[0].total := 300.0, [1724].log_data[0].time := 300.0, [1724].log_data[0].minminute := 10, [1724].log_data[0].maxminute := 10, [1724].log_data[0].valid := 1, [1724].log_data[1].valid := 1, [1724].log_data[2].valid := 1, [1724].log_data[3].valid := 1, [1724].log_data[4].valid := 1, [1724].time.Year := 2022, [1724].time.Month := 4, [1724].time.Day := 29, [1724].time.Hour := 21, [1724].time.Minute := 14, [1724].time.Second := 59, [1724].time.DST_ON := 1, [1725].log_data[0].min := 1.0, [1725].log_data[0].max := 1.0, [1725].log_data[0].total := 300.0, [1725].log_data[0].time := 300.0, [1725].log_data[0].minminute := 15, [1725].log_data[0].maxminute := 15, [1725].log_data[0].valid := 1, [1725].log_data[1].valid := 1, [1725].log_data[2].valid := 1, [1725].log_data[3].valid := 1, [1725].log_data[4].valid := 1, [1725].time.Year := 2022, [1725].time.Month := 4, [1725].time.Day := 29, [1725].time.Hour := 21, [1725].time.Minute := 19, [1725].time.Second := 59, [1725].time.DST_ON := 1, [1726].log_data[0].min := 1.0, [1726].log_data[0].max := 1.0, [1726].log_data[0].total := 300.0, [1726].log_data[0].time := 300.0, [1726].log_data[0].minminute := 20, [1726].log_data[0].maxminute := 20, [1726].log_data[0].valid := 1,
        [1726].log_data[1].valid := 1, [1726].log_data[2].valid := 1, [1726].log_data[3].valid := 1, [1726].log_data[4].valid := 1, [1726].time.Year := 2022, [1726].time.Month := 4, [1726].time.Day := 29, [1726].time.Hour := 21, [1726].time.Minute := 24, [1726].time.Second := 59, [1726].time.DST_ON := 1, [1727].log_data[0].min := 1.0, [1727].log_data[0].max := 1.0, [1727].log_data[0].total := 300.0, [1727].log_data[0].time := 300.0, [1727].log_data[0].minminute := 25, [1727].log_data[0].maxminute := 25, [1727].log_data[0].valid := 1, [1727].log_data[1].valid := 1, [1727].log_data[2].valid := 1, [1727].log_data[3].valid := 1, [1727].log_data[4].valid := 1, [1727].time.Year := 2022, [1727].time.Month := 4, [1727].time.Day := 29, [1727].time.Hour := 21, [1727].time.Minute := 29, [1727].time.Second := 59, [1727].time.DST_ON := 1, [1728].log_data[0].min := 1.0, [1728].log_data[0].max := 1.0, [1728].log_data[0].total := 300.0, [1728].log_data[0].time := 300.0, [1728].log_data[0].minminute := 30, [1728].log_data[0].maxminute := 30, [1728].log_data[0].valid := 1, [1728].log_data[1].valid := 1, [1728].log_data[2].valid := 1, [1728].log_data[3].valid := 1, [1728].log_data[4].valid := 1, [1728].time.Year := 2022, [1728].time.Month := 4, [1728].time.Day := 29, [1728].time.Hour := 21, [1728].time.Minute := 34, [1728].time.Second := 59, [1728].time.DST_ON := 1, [1729].log_data[0].min := 1.0, [1729].log_data[0].max := 1.0, [1729].log_data[0].total := 300.0, [1729].log_data[0].time := 300.0, [1729].log_data[0].minminute := 35, [1729].log_data[0].maxminute := 35, [1729].log_data[0].valid := 1, [1729].log_data[1].valid := 1, [1729].log_data[2].valid := 1, [1729].log_data[3].valid := 1, [1729].log_data[4].valid := 1, [1729].time.Year := 2022, [1729].time.Month := 4,
        [1729].time.Day := 29, [1729].time.Hour := 21, [1729].time.Minute := 39, [1729].time.Second := 59, [1729].time.DST_ON := 1, [1730].log_data[0].min := 1.0, [1730].log_data[0].max := 1.0, [1730].log_data[0].total := 300.0, [1730].log_data[0].time := 300.0, [1730].log_data[0].minminute := 40, [1730].log_data[0].maxminute := 40, [1730].log_data[0].valid := 1, [1730].log_data[1].valid := 1, [1730].log_data[2].valid := 1, [1730].log_data[3].valid := 1, [1730].log_data[4].valid := 1, [1730].time.Year := 2022, [1730].time.Month := 4, [1730].time.Day := 29, [1730].time.Hour := 21, [1730].time.Minute := 44, [1730].time.Second := 59, [1730].time.DST_ON := 1, [1731].log_data[0].min := 1.0, [1731].log_data[0].max := 1.0, [1731].log_data[0].total := 300.0, [1731].log_data[0].time := 300.0, [1731].log_data[0].minminute := 45, [1731].log_data[0].maxminute := 45, [1731].log_data[0].valid := 1, [1731].log_data[1].valid := 1, [1731].log_data[2].valid := 1, [1731].log_data[3].valid := 1, [1731].log_data[4].valid := 1, [1731].time.Year := 2022, [1731].time.Month := 4, [1731].time.Day := 29, [1731].time.Hour := 21, [1731].time.Minute := 49, [1731].time.Second := 59, [1731].time.DST_ON := 1, [1732].log_data[0].min := 1.0, [1732].log_data[0].max := 1.0, [1732].log_data[0].total := 300.0, [1732].log_data[0].time := 300.0, [1732].log_data[0].minminute := 50, [1732].log_data[0].maxminute := 50, [1732].log_data[0].valid := 1, [1732].log_data[1].valid := 1, [1732].log_data[2].valid := 1, [1732].log_data[3].valid := 1, [1732].log_data[4].valid := 1, [1732].time.Year := 2022, [1732].time.Month := 4, [1732].time.Day := 29, [1732].time.Hour := 21, [1732].time.Minute := 54, [1732].time.Second := 59, [1732].time.DST_ON := 1, [1733].log_data[0].min := 1.0,
        [1733].log_data[0].max := 1.0, [1733].log_data[0].total := 300.0, [1733].log_data[0].time := 300.0, [1733].log_data[0].minminute := 55, [1733].log_data[0].maxminute := 55, [1733].log_data[0].valid := 1, [1733].log_data[1].valid := 1, [1733].log_data[2].valid := 1, [1733].log_data[3].valid := 1, [1733].log_data[4].valid := 1, [1733].time.Year := 2022, [1733].time.Month := 4, [1733].time.Day := 29, [1733].time.Hour := 21, [1733].time.Minute := 59, [1733].time.Second := 59, [1733].time.DST_ON := 1, [1734].log_data[0].min := 1.0, [1734].log_data[0].max := 1.0, [1734].log_data[0].total := 300.0, [1734].log_data[0].time := 300.0, [1734].log_data[0].valid := 1, [1734].log_data[1].valid := 1, [1734].log_data[2].valid := 1, [1734].log_data[3].valid := 1, [1734].log_data[4].valid := 1, [1734].time.Year := 2022, [1734].time.Month := 4, [1734].time.Day := 29, [1734].time.Hour := 22, [1734].time.Minute := 4, [1734].time.Second := 59, [1734].time.DST_ON := 1, [1735].log_data[0].min := 1.0, [1735].log_data[0].max := 1.0, [1735].log_data[0].total := 300.0, [1735].log_data[0].time := 300.0, [1735].log_data[0].minminute := 5, [1735].log_data[0].maxminute := 5, [1735].log_data[0].valid := 1, [1735].log_data[1].valid := 1, [1735].log_data[2].valid := 1, [1735].log_data[3].valid := 1, [1735].log_data[4].valid := 1, [1735].time.Year := 2022, [1735].time.Month := 4, [1735].time.Day := 29, [1735].time.Hour := 22, [1735].time.Minute := 9, [1735].time.Second := 59, [1735].time.DST_ON := 1, [1736].log_data[0].min := 1.0, [1736].log_data[0].max := 1.0, [1736].log_data[0].total := 300.0, [1736].log_data[0].time := 300.0, [1736].log_data[0].minminute := 10, [1736].log_data[0].maxminute := 10, [1736].log_data[0].valid := 1, [1736].log_data[1].valid := 1, [1736].log_data[2].valid := 1,
        [1736].log_data[3].valid := 1, [1736].log_data[4].valid := 1, [1736].time.Year := 2022, [1736].time.Month := 4, [1736].time.Day := 29, [1736].time.Hour := 22, [1736].time.Minute := 14, [1736].time.Second := 59, [1736].time.DST_ON := 1, [1737].log_data[0].min := 1.0, [1737].log_data[0].max := 1.0, [1737].log_data[0].total := 300.0, [1737].log_data[0].time := 300.0, [1737].log_data[0].minminute := 15, [1737].log_data[0].maxminute := 15, [1737].log_data[0].valid := 1, [1737].log_data[1].valid := 1, [1737].log_data[2].valid := 1, [1737].log_data[3].valid := 1, [1737].log_data[4].valid := 1, [1737].time.Year := 2022, [1737].time.Month := 4, [1737].time.Day := 29, [1737].time.Hour := 22, [1737].time.Minute := 19, [1737].time.Second := 59, [1737].time.DST_ON := 1, [1738].log_data[0].min := 1.0, [1738].log_data[0].max := 1.0, [1738].log_data[0].total := 300.0, [1738].log_data[0].time := 300.0, [1738].log_data[0].minminute := 20, [1738].log_data[0].maxminute := 20, [1738].log_data[0].valid := 1, [1738].log_data[1].valid := 1, [1738].log_data[2].valid := 1, [1738].log_data[3].valid := 1, [1738].log_data[4].valid := 1, [1738].time.Year := 2022, [1738].time.Month := 4, [1738].time.Day := 29, [1738].time.Hour := 22, [1738].time.Minute := 24, [1738].time.Second := 59, [1738].time.DST_ON := 1, [1739].log_data[0].min := 1.0, [1739].log_data[0].max := 1.0, [1739].log_data[0].total := 300.0, [1739].log_data[0].time := 300.0, [1739].log_data[0].minminute := 25, [1739].log_data[0].maxminute := 25, [1739].log_data[0].valid := 1, [1739].log_data[1].valid := 1, [1739].log_data[2].valid := 1, [1739].log_data[3].valid := 1, [1739].log_data[4].valid := 1, [1739].time.Year := 2022, [1739].time.Month := 4, [1739].time.Day := 29, [1739].time.Hour := 22,
        [1739].time.Minute := 29, [1739].time.Second := 59, [1739].time.DST_ON := 1, [1740].log_data[0].min := 1.0, [1740].log_data[0].max := 1.0, [1740].log_data[0].total := 300.0, [1740].log_data[0].time := 300.0, [1740].log_data[0].minminute := 30, [1740].log_data[0].maxminute := 30, [1740].log_data[0].valid := 1, [1740].log_data[1].valid := 1, [1740].log_data[2].valid := 1, [1740].log_data[3].valid := 1, [1740].log_data[4].valid := 1, [1740].time.Year := 2022, [1740].time.Month := 4, [1740].time.Day := 29, [1740].time.Hour := 22, [1740].time.Minute := 34, [1740].time.Second := 59, [1740].time.DST_ON := 1, [1741].log_data[0].min := 1.0, [1741].log_data[0].max := 1.0, [1741].log_data[0].total := 300.0, [1741].log_data[0].time := 300.0, [1741].log_data[0].minminute := 35, [1741].log_data[0].maxminute := 35, [1741].log_data[0].valid := 1, [1741].log_data[1].valid := 1, [1741].log_data[2].valid := 1, [1741].log_data[3].valid := 1, [1741].log_data[4].valid := 1, [1741].time.Year := 2022, [1741].time.Month := 4, [1741].time.Day := 29, [1741].time.Hour := 22, [1741].time.Minute := 39, [1741].time.Second := 59, [1741].time.DST_ON := 1, [1742].log_data[0].min := 1.0, [1742].log_data[0].max := 1.0, [1742].log_data[0].total := 300.0, [1742].log_data[0].time := 300.0, [1742].log_data[0].minminute := 40, [1742].log_data[0].maxminute := 40, [1742].log_data[0].valid := 1, [1742].log_data[1].valid := 1, [1742].log_data[2].valid := 1, [1742].log_data[3].valid := 1, [1742].log_data[4].valid := 1, [1742].time.Year := 2022, [1742].time.Month := 4, [1742].time.Day := 29, [1742].time.Hour := 22, [1742].time.Minute := 44, [1742].time.Second := 59, [1742].time.DST_ON := 1, [1743].log_data[0].min := 1.0, [1743].log_data[0].max := 1.0, [1743].log_data[0].total := 300.0,
        [1743].log_data[0].time := 300.0, [1743].log_data[0].minminute := 45, [1743].log_data[0].maxminute := 45, [1743].log_data[0].valid := 1, [1743].log_data[1].valid := 1, [1743].log_data[2].valid := 1, [1743].log_data[3].valid := 1, [1743].log_data[4].valid := 1, [1743].time.Year := 2022, [1743].time.Month := 4, [1743].time.Day := 29, [1743].time.Hour := 22, [1743].time.Minute := 49, [1743].time.Second := 59, [1743].time.DST_ON := 1, [1744].log_data[0].min := 1.0, [1744].log_data[0].max := 1.0, [1744].log_data[0].total := 300.0, [1744].log_data[0].time := 300.0, [1744].log_data[0].minminute := 50, [1744].log_data[0].maxminute := 50, [1744].log_data[0].valid := 1, [1744].log_data[1].valid := 1, [1744].log_data[2].valid := 1, [1744].log_data[3].valid := 1, [1744].log_data[4].valid := 1, [1744].time.Year := 2022, [1744].time.Month := 4, [1744].time.Day := 29, [1744].time.Hour := 22, [1744].time.Minute := 54, [1744].time.Second := 59, [1744].time.DST_ON := 1, [1745].log_data[0].min := 1.0, [1745].log_data[0].max := 1.0, [1745].log_data[0].total := 300.0, [1745].log_data[0].time := 300.0, [1745].log_data[0].minminute := 55, [1745].log_data[0].maxminute := 55, [1745].log_data[0].valid := 1, [1745].log_data[1].valid := 1, [1745].log_data[2].valid := 1, [1745].log_data[3].valid := 1, [1745].log_data[4].valid := 1, [1745].time.Year := 2022, [1745].time.Month := 4, [1745].time.Day := 29, [1745].time.Hour := 22, [1745].time.Minute := 59, [1745].time.Second := 59, [1745].time.DST_ON := 1, [1746].log_data[0].min := 1.0, [1746].log_data[0].max := 1.0, [1746].log_data[0].total := 300.0, [1746].log_data[0].time := 300.0, [1746].log_data[0].valid := 1, [1746].log_data[1].valid := 1, [1746].log_data[2].valid := 1, [1746].log_data[3].valid := 1, [1746].log_data[4].valid := 1,
        [1746].time.Year := 2022, [1746].time.Month := 4, [1746].time.Day := 29, [1746].time.Hour := 23, [1746].time.Minute := 4, [1746].time.Second := 59, [1746].time.DST_ON := 1, [1747].log_data[0].min := 1.0, [1747].log_data[0].max := 1.0, [1747].log_data[0].total := 300.0, [1747].log_data[0].time := 300.0, [1747].log_data[0].minminute := 5, [1747].log_data[0].maxminute := 5, [1747].log_data[0].valid := 1, [1747].log_data[1].valid := 1, [1747].log_data[2].valid := 1, [1747].log_data[3].valid := 1, [1747].log_data[4].valid := 1, [1747].time.Year := 2022, [1747].time.Month := 4, [1747].time.Day := 29, [1747].time.Hour := 23, [1747].time.Minute := 9, [1747].time.Second := 59, [1747].time.DST_ON := 1, [1748].log_data[0].min := 1.0, [1748].log_data[0].max := 1.0, [1748].log_data[0].total := 300.0, [1748].log_data[0].time := 300.0, [1748].log_data[0].minminute := 10, [1748].log_data[0].maxminute := 10, [1748].log_data[0].valid := 1, [1748].log_data[1].valid := 1, [1748].log_data[2].valid := 1, [1748].log_data[3].valid := 1, [1748].log_data[4].valid := 1, [1748].time.Year := 2022, [1748].time.Month := 4, [1748].time.Day := 29, [1748].time.Hour := 23, [1748].time.Minute := 14, [1748].time.Second := 59, [1748].time.DST_ON := 1, [1749].log_data[0].min := 1.0, [1749].log_data[0].max := 1.0, [1749].log_data[0].total := 300.0, [1749].log_data[0].time := 300.0, [1749].log_data[0].minminute := 15, [1749].log_data[0].maxminute := 15, [1749].log_data[0].valid := 1, [1749].log_data[1].valid := 1, [1749].log_data[2].valid := 1, [1749].log_data[3].valid := 1, [1749].log_data[4].valid := 1, [1749].time.Year := 2022, [1749].time.Month := 4, [1749].time.Day := 29, [1749].time.Hour := 23, [1749].time.Minute := 19, [1749].time.Second := 59,
        [1749].time.DST_ON := 1, [1750].log_data[0].min := 1.0, [1750].log_data[0].max := 1.0, [1750].log_data[0].total := 300.0, [1750].log_data[0].time := 300.0, [1750].log_data[0].minminute := 20, [1750].log_data[0].maxminute := 20, [1750].log_data[0].valid := 1, [1750].log_data[1].valid := 1, [1750].log_data[2].valid := 1, [1750].log_data[3].valid := 1, [1750].log_data[4].valid := 1, [1750].time.Year := 2022, [1750].time.Month := 4, [1750].time.Day := 29, [1750].time.Hour := 23, [1750].time.Minute := 24, [1750].time.Second := 59, [1750].time.DST_ON := 1, [1751].log_data[0].min := 1.0, [1751].log_data[0].max := 1.0, [1751].log_data[0].total := 300.0, [1751].log_data[0].time := 300.0, [1751].log_data[0].minminute := 25, [1751].log_data[0].maxminute := 25, [1751].log_data[0].valid := 1, [1751].log_data[1].valid := 1, [1751].log_data[2].valid := 1, [1751].log_data[3].valid := 1, [1751].log_data[4].valid := 1, [1751].time.Year := 2022, [1751].time.Month := 4, [1751].time.Day := 29, [1751].time.Hour := 23, [1751].time.Minute := 29, [1751].time.Second := 59, [1751].time.DST_ON := 1, [1752].log_data[0].min := 1.0, [1752].log_data[0].max := 1.0, [1752].log_data[0].total := 300.0, [1752].log_data[0].time := 300.0, [1752].log_data[0].minminute := 30, [1752].log_data[0].maxminute := 30, [1752].log_data[0].valid := 1, [1752].log_data[1].valid := 1, [1752].log_data[2].valid := 1, [1752].log_data[3].valid := 1, [1752].log_data[4].valid := 1, [1752].time.Year := 2022, [1752].time.Month := 4, [1752].time.Day := 29, [1752].time.Hour := 23, [1752].time.Minute := 34, [1752].time.Second := 59, [1752].time.DST_ON := 1, [1753].log_data[0].min := 1.0, [1753].log_data[0].max := 1.0, [1753].log_data[0].total := 300.0, [1753].log_data[0].time := 300.0, [1753].log_data[0].minminute := 35,
        [1753].log_data[0].maxminute := 35, [1753].log_data[0].valid := 1, [1753].log_data[1].valid := 1, [1753].log_data[2].valid := 1, [1753].log_data[3].valid := 1, [1753].log_data[4].valid := 1, [1753].time.Year := 2022, [1753].time.Month := 4, [1753].time.Day := 29, [1753].time.Hour := 23, [1753].time.Minute := 39, [1753].time.Second := 59, [1753].time.DST_ON := 1, [1754].log_data[0].min := 1.0, [1754].log_data[0].max := 1.0, [1754].log_data[0].total := 300.0, [1754].log_data[0].time := 300.0, [1754].log_data[0].minminute := 40, [1754].log_data[0].maxminute := 40, [1754].log_data[0].valid := 1, [1754].log_data[1].valid := 1, [1754].log_data[2].valid := 1, [1754].log_data[3].valid := 1, [1754].log_data[4].valid := 1, [1754].time.Year := 2022, [1754].time.Month := 4, [1754].time.Day := 29, [1754].time.Hour := 23, [1754].time.Minute := 44, [1754].time.Second := 59, [1754].time.DST_ON := 1, [1755].log_data[0].min := 1.0, [1755].log_data[0].max := 1.0, [1755].log_data[0].total := 300.0, [1755].log_data[0].time := 300.0, [1755].log_data[0].minminute := 45, [1755].log_data[0].maxminute := 45, [1755].log_data[0].valid := 1, [1755].log_data[1].valid := 1, [1755].log_data[2].valid := 1, [1755].log_data[3].valid := 1, [1755].log_data[4].valid := 1, [1755].time.Year := 2022, [1755].time.Month := 4, [1755].time.Day := 29, [1755].time.Hour := 23, [1755].time.Minute := 49, [1755].time.Second := 59, [1755].time.DST_ON := 1, [1756].log_data[0].min := 1.0, [1756].log_data[0].max := 1.0, [1756].log_data[0].total := 300.0, [1756].log_data[0].time := 300.0, [1756].log_data[0].minminute := 50, [1756].log_data[0].maxminute := 50, [1756].log_data[0].valid := 1, [1756].log_data[1].valid := 1, [1756].log_data[2].valid := 1, [1756].log_data[3].valid := 1, [1756].log_data[4].valid := 1,
        [1756].time.Year := 2022, [1756].time.Month := 4, [1756].time.Day := 29, [1756].time.Hour := 23, [1756].time.Minute := 54, [1756].time.Second := 59, [1756].time.DST_ON := 1, [1757].log_data[0].min := 1.0, [1757].log_data[0].max := 1.0, [1757].log_data[0].total := 300.0, [1757].log_data[0].time := 300.0, [1757].log_data[0].minminute := 55, [1757].log_data[0].maxminute := 55, [1757].log_data[0].valid := 1, [1757].log_data[1].valid := 1, [1757].log_data[2].valid := 1, [1757].log_data[3].valid := 1, [1757].log_data[4].valid := 1, [1757].time.Year := 2022, [1757].time.Month := 4, [1757].time.Day := 29, [1757].time.Hour := 23, [1757].time.Minute := 59, [1757].time.Second := 59, [1757].time.DST_ON := 1, [1758].log_data[0].min := 1.0, [1758].log_data[0].max := 1.0, [1758].log_data[0].total := 300.0, [1758].log_data[0].time := 300.0, [1758].log_data[0].valid := 1, [1758].log_data[1].valid := 1, [1758].log_data[2].valid := 1, [1758].log_data[3].valid := 1, [1758].log_data[4].valid := 1, [1758].time.Year := 2022, [1758].time.Month := 4, [1758].time.Day := 30, [1758].time.Minute := 4, [1758].time.Second := 59, [1758].time.DST_ON := 1, [1759].log_data[0].min := 1.0, [1759].log_data[0].max := 1.0, [1759].log_data[0].total := 300.0, [1759].log_data[0].time := 300.0, [1759].log_data[0].minminute := 5, [1759].log_data[0].maxminute := 5, [1759].log_data[0].valid := 1, [1759].log_data[1].valid := 1, [1759].log_data[2].valid := 1, [1759].log_data[3].valid := 1, [1759].log_data[4].valid := 1, [1759].time.Year := 2022, [1759].time.Month := 4, [1759].time.Day := 30, [1759].time.Minute := 9, [1759].time.Second := 59, [1759].time.DST_ON := 1, [1760].log_data[0].min := 1.0, [1760].log_data[0].max := 1.0, [1760].log_data[0].total := 300.0,
        [1760].log_data[0].time := 300.0, [1760].log_data[0].minminute := 10, [1760].log_data[0].maxminute := 10, [1760].log_data[0].valid := 1, [1760].log_data[1].valid := 1, [1760].log_data[2].valid := 1, [1760].log_data[3].valid := 1, [1760].log_data[4].valid := 1, [1760].time.Year := 2022, [1760].time.Month := 4, [1760].time.Day := 30, [1760].time.Minute := 14, [1760].time.Second := 59, [1760].time.DST_ON := 1, [1761].log_data[0].min := 1.0, [1761].log_data[0].max := 1.0, [1761].log_data[0].total := 300.0, [1761].log_data[0].time := 300.0, [1761].log_data[0].minminute := 15, [1761].log_data[0].maxminute := 15, [1761].log_data[0].valid := 1, [1761].log_data[1].valid := 1, [1761].log_data[2].valid := 1, [1761].log_data[3].valid := 1, [1761].log_data[4].valid := 1, [1761].time.Year := 2022, [1761].time.Month := 4, [1761].time.Day := 30, [1761].time.Minute := 19, [1761].time.Second := 59, [1761].time.DST_ON := 1, [1762].log_data[0].min := 1.0, [1762].log_data[0].max := 1.0, [1762].log_data[0].total := 300.0, [1762].log_data[0].time := 300.0, [1762].log_data[0].minminute := 20, [1762].log_data[0].maxminute := 20, [1762].log_data[0].valid := 1, [1762].log_data[1].valid := 1, [1762].log_data[2].valid := 1, [1762].log_data[3].valid := 1, [1762].log_data[4].valid := 1, [1762].time.Year := 2022, [1762].time.Month := 4, [1762].time.Day := 30, [1762].time.Minute := 24, [1762].time.Second := 59, [1762].time.DST_ON := 1, [1763].log_data[0].min := 1.0, [1763].log_data[0].max := 1.0, [1763].log_data[0].total := 300.0, [1763].log_data[0].time := 300.0, [1763].log_data[0].minminute := 25, [1763].log_data[0].maxminute := 25, [1763].log_data[0].valid := 1, [1763].log_data[1].valid := 1, [1763].log_data[2].valid := 1, [1763].log_data[3].valid := 1, [1763].log_data[4].valid := 1, [1763].time.Year := 2022,
        [1763].time.Month := 4, [1763].time.Day := 30, [1763].time.Minute := 29, [1763].time.Second := 59, [1763].time.DST_ON := 1, [1764].log_data[0].min := 1.0, [1764].log_data[0].max := 1.0, [1764].log_data[0].total := 300.0, [1764].log_data[0].time := 300.0, [1764].log_data[0].minminute := 30, [1764].log_data[0].maxminute := 30, [1764].log_data[0].valid := 1, [1764].log_data[1].valid := 1, [1764].log_data[2].valid := 1, [1764].log_data[3].valid := 1, [1764].log_data[4].valid := 1, [1764].time.Year := 2022, [1764].time.Month := 4, [1764].time.Day := 30, [1764].time.Minute := 34, [1764].time.Second := 59, [1764].time.DST_ON := 1, [1765].log_data[0].min := 1.0, [1765].log_data[0].max := 1.0, [1765].log_data[0].total := 300.0, [1765].log_data[0].time := 300.0, [1765].log_data[0].minminute := 35, [1765].log_data[0].maxminute := 35, [1765].log_data[0].valid := 1, [1765].log_data[1].valid := 1, [1765].log_data[2].valid := 1, [1765].log_data[3].valid := 1, [1765].log_data[4].valid := 1, [1765].time.Year := 2022, [1765].time.Month := 4, [1765].time.Day := 30, [1765].time.Minute := 39, [1765].time.Second := 59, [1765].time.DST_ON := 1, [1766].log_data[0].min := 1.0, [1766].log_data[0].max := 1.0, [1766].log_data[0].total := 300.0, [1766].log_data[0].time := 300.0, [1766].log_data[0].minminute := 40, [1766].log_data[0].maxminute := 40, [1766].log_data[0].valid := 1, [1766].log_data[1].valid := 1, [1766].log_data[2].valid := 1, [1766].log_data[3].valid := 1, [1766].log_data[4].valid := 1, [1766].time.Year := 2022, [1766].time.Month := 4, [1766].time.Day := 30, [1766].time.Minute := 44, [1766].time.Second := 59, [1766].time.DST_ON := 1, [1767].log_data[0].min := 1.0, [1767].log_data[0].max := 1.0, [1767].log_data[0].total := 300.0, [1767].log_data[0].time := 300.0,
        [1767].log_data[0].minminute := 45, [1767].log_data[0].maxminute := 45, [1767].log_data[0].valid := 1, [1767].log_data[1].valid := 1, [1767].log_data[2].valid := 1, [1767].log_data[3].valid := 1, [1767].log_data[4].valid := 1, [1767].time.Year := 2022, [1767].time.Month := 4, [1767].time.Day := 30, [1767].time.Minute := 49, [1767].time.Second := 59, [1767].time.DST_ON := 1, [1768].log_data[0].min := 1.0, [1768].log_data[0].max := 1.0, [1768].log_data[0].total := 300.0, [1768].log_data[0].time := 300.0, [1768].log_data[0].minminute := 50, [1768].log_data[0].maxminute := 50, [1768].log_data[0].valid := 1, [1768].log_data[1].valid := 1, [1768].log_data[2].valid := 1, [1768].log_data[3].valid := 1, [1768].log_data[4].valid := 1, [1768].time.Year := 2022, [1768].time.Month := 4, [1768].time.Day := 30, [1768].time.Minute := 54, [1768].time.Second := 59, [1768].time.DST_ON := 1, [1769].log_data[0].min := 1.0, [1769].log_data[0].max := 1.0, [1769].log_data[0].total := 300.0, [1769].log_data[0].time := 300.0, [1769].log_data[0].minminute := 55, [1769].log_data[0].maxminute := 55, [1769].log_data[0].valid := 1, [1769].log_data[1].valid := 1, [1769].log_data[2].valid := 1, [1769].log_data[3].valid := 1, [1769].log_data[4].valid := 1, [1769].time.Year := 2022, [1769].time.Month := 4, [1769].time.Day := 30, [1769].time.Minute := 59, [1769].time.Second := 59, [1769].time.DST_ON := 1, [1770].log_data[0].min := 1.0, [1770].log_data[0].max := 1.0, [1770].log_data[0].total := 300.0, [1770].log_data[0].time := 300.0, [1770].log_data[0].valid := 1, [1770].log_data[1].valid := 1, [1770].log_data[2].valid := 1, [1770].log_data[3].valid := 1, [1770].log_data[4].valid := 1, [1770].time.Year := 2022, [1770].time.Month := 4, [1770].time.Day := 30, [1770].time.Hour := 1,
        [1770].time.Minute := 4, [1770].time.Second := 59, [1770].time.DST_ON := 1, [1771].log_data[0].min := 1.0, [1771].log_data[0].max := 1.0, [1771].log_data[0].total := 300.0, [1771].log_data[0].time := 300.0, [1771].log_data[0].minminute := 5, [1771].log_data[0].maxminute := 5, [1771].log_data[0].valid := 1, [1771].log_data[1].valid := 1, [1771].log_data[2].valid := 1, [1771].log_data[3].valid := 1, [1771].log_data[4].valid := 1, [1771].time.Year := 2022, [1771].time.Month := 4, [1771].time.Day := 30, [1771].time.Hour := 1, [1771].time.Minute := 9, [1771].time.Second := 59, [1771].time.DST_ON := 1, [1772].log_data[0].min := 1.0, [1772].log_data[0].max := 1.0, [1772].log_data[0].total := 300.0, [1772].log_data[0].time := 300.0, [1772].log_data[0].minminute := 10, [1772].log_data[0].maxminute := 10, [1772].log_data[0].valid := 1, [1772].log_data[1].valid := 1, [1772].log_data[2].valid := 1, [1772].log_data[3].valid := 1, [1772].log_data[4].valid := 1, [1772].time.Year := 2022, [1772].time.Month := 4, [1772].time.Day := 30, [1772].time.Hour := 1, [1772].time.Minute := 14, [1772].time.Second := 59, [1772].time.DST_ON := 1, [1773].log_data[0].min := 1.0, [1773].log_data[0].max := 1.0, [1773].log_data[0].total := 300.0, [1773].log_data[0].time := 300.0, [1773].log_data[0].minminute := 15, [1773].log_data[0].maxminute := 15, [1773].log_data[0].valid := 1, [1773].log_data[1].valid := 1, [1773].log_data[2].valid := 1, [1773].log_data[3].valid := 1, [1773].log_data[4].valid := 1, [1773].time.Year := 2022, [1773].time.Month := 4, [1773].time.Day := 30, [1773].time.Hour := 1, [1773].time.Minute := 19, [1773].time.Second := 59, [1773].time.DST_ON := 1, [1774].log_data[0].min := 1.0, [1774].log_data[0].max := 1.0, [1774].log_data[0].total := 300.0,
        [1774].log_data[0].time := 300.0, [1774].log_data[0].minminute := 20, [1774].log_data[0].maxminute := 20, [1774].log_data[0].valid := 1, [1774].log_data[1].valid := 1, [1774].log_data[2].valid := 1, [1774].log_data[3].valid := 1, [1774].log_data[4].valid := 1, [1774].time.Year := 2022, [1774].time.Month := 4, [1774].time.Day := 30, [1774].time.Hour := 1, [1774].time.Minute := 24, [1774].time.Second := 59, [1774].time.DST_ON := 1, [1775].log_data[0].min := 1.0, [1775].log_data[0].max := 1.0, [1775].log_data[0].total := 300.0, [1775].log_data[0].time := 300.0, [1775].log_data[0].minminute := 25, [1775].log_data[0].maxminute := 25, [1775].log_data[0].valid := 1, [1775].log_data[1].valid := 1, [1775].log_data[2].valid := 1, [1775].log_data[3].valid := 1, [1775].log_data[4].valid := 1, [1775].time.Year := 2022, [1775].time.Month := 4, [1775].time.Day := 30, [1775].time.Hour := 1, [1775].time.Minute := 29, [1775].time.Second := 59, [1775].time.DST_ON := 1, [1776].log_data[0].min := 1.0, [1776].log_data[0].max := 1.0, [1776].log_data[0].total := 300.0, [1776].log_data[0].time := 300.0, [1776].log_data[0].minminute := 30, [1776].log_data[0].maxminute := 30, [1776].log_data[0].valid := 1, [1776].log_data[1].valid := 1, [1776].log_data[2].valid := 1, [1776].log_data[3].valid := 1, [1776].log_data[4].valid := 1, [1776].time.Year := 2022, [1776].time.Month := 4, [1776].time.Day := 30, [1776].time.Hour := 1, [1776].time.Minute := 34, [1776].time.Second := 59, [1776].time.DST_ON := 1, [1777].log_data[0].min := 1.0, [1777].log_data[0].max := 1.0, [1777].log_data[0].total := 300.0, [1777].log_data[0].time := 300.0, [1777].log_data[0].minminute := 35, [1777].log_data[0].maxminute := 35, [1777].log_data[0].valid := 1, [1777].log_data[1].valid := 1, [1777].log_data[2].valid := 1,
        [1777].log_data[3].valid := 1, [1777].log_data[4].valid := 1, [1777].time.Year := 2022, [1777].time.Month := 4, [1777].time.Day := 30, [1777].time.Hour := 1, [1777].time.Minute := 39, [1777].time.Second := 59, [1777].time.DST_ON := 1, [1778].log_data[0].min := 1.0, [1778].log_data[0].max := 1.0, [1778].log_data[0].total := 300.0, [1778].log_data[0].time := 300.0, [1778].log_data[0].minminute := 40, [1778].log_data[0].maxminute := 40, [1778].log_data[0].valid := 1, [1778].log_data[1].valid := 1, [1778].log_data[2].valid := 1, [1778].log_data[3].valid := 1, [1778].log_data[4].valid := 1, [1778].time.Year := 2022, [1778].time.Month := 4, [1778].time.Day := 30, [1778].time.Hour := 1, [1778].time.Minute := 44, [1778].time.Second := 59, [1778].time.DST_ON := 1, [1779].log_data[0].min := 1.0, [1779].log_data[0].max := 1.0, [1779].log_data[0].total := 300.0, [1779].log_data[0].time := 300.0, [1779].log_data[0].minminute := 45, [1779].log_data[0].maxminute := 45, [1779].log_data[0].valid := 1, [1779].log_data[1].valid := 1, [1779].log_data[2].valid := 1, [1779].log_data[3].valid := 1, [1779].log_data[4].valid := 1, [1779].time.Year := 2022, [1779].time.Month := 4, [1779].time.Day := 30, [1779].time.Hour := 1, [1779].time.Minute := 49, [1779].time.Second := 59, [1779].time.DST_ON := 1, [1780].log_data[0].min := 1.0, [1780].log_data[0].max := 1.0, [1780].log_data[0].total := 300.0, [1780].log_data[0].time := 300.0, [1780].log_data[0].minminute := 50, [1780].log_data[0].maxminute := 50, [1780].log_data[0].valid := 1, [1780].log_data[1].valid := 1, [1780].log_data[2].valid := 1, [1780].log_data[3].valid := 1, [1780].log_data[4].valid := 1, [1780].time.Year := 2022, [1780].time.Month := 4, [1780].time.Day := 30, [1780].time.Hour := 1,
        [1780].time.Minute := 54, [1780].time.Second := 59, [1780].time.DST_ON := 1, [1781].log_data[0].min := 1.0, [1781].log_data[0].max := 1.0, [1781].log_data[0].total := 300.0, [1781].log_data[0].time := 300.0, [1781].log_data[0].minminute := 55, [1781].log_data[0].maxminute := 55, [1781].log_data[0].valid := 1, [1781].log_data[1].valid := 1, [1781].log_data[2].valid := 1, [1781].log_data[3].valid := 1, [1781].log_data[4].valid := 1, [1781].time.Year := 2022, [1781].time.Month := 4, [1781].time.Day := 30, [1781].time.Hour := 1, [1781].time.Minute := 59, [1781].time.Second := 59, [1781].time.DST_ON := 1, [1782].log_data[0].min := 1.0, [1782].log_data[0].max := 1.0, [1782].log_data[0].total := 300.0, [1782].log_data[0].time := 300.0, [1782].log_data[0].valid := 1, [1782].log_data[1].valid := 1, [1782].log_data[2].valid := 1, [1782].log_data[3].valid := 1, [1782].log_data[4].valid := 1, [1782].time.Year := 2022, [1782].time.Month := 4, [1782].time.Day := 30, [1782].time.Hour := 2, [1782].time.Minute := 4, [1782].time.Second := 59, [1782].time.DST_ON := 1, [1783].log_data[0].min := 1.0, [1783].log_data[0].max := 1.0, [1783].log_data[0].total := 300.0, [1783].log_data[0].time := 300.0, [1783].log_data[0].minminute := 5, [1783].log_data[0].maxminute := 5, [1783].log_data[0].valid := 1, [1783].log_data[1].valid := 1, [1783].log_data[2].valid := 1, [1783].log_data[3].valid := 1, [1783].log_data[4].valid := 1, [1783].time.Year := 2022, [1783].time.Month := 4, [1783].time.Day := 30, [1783].time.Hour := 2, [1783].time.Minute := 9, [1783].time.Second := 59, [1783].time.DST_ON := 1, [1784].log_data[0].min := 1.0, [1784].log_data[0].max := 1.0, [1784].log_data[0].total := 300.0, [1784].log_data[0].time := 300.0, [1784].log_data[0].minminute := 10,
        [1784].log_data[0].maxminute := 10, [1784].log_data[0].valid := 1, [1784].log_data[1].valid := 1, [1784].log_data[2].valid := 1, [1784].log_data[3].valid := 1, [1784].log_data[4].valid := 1, [1784].time.Year := 2022, [1784].time.Month := 4, [1784].time.Day := 30, [1784].time.Hour := 2, [1784].time.Minute := 14, [1784].time.Second := 59, [1784].time.DST_ON := 1, [1785].log_data[0].min := 1.0, [1785].log_data[0].max := 1.0, [1785].log_data[0].total := 300.0, [1785].log_data[0].time := 300.0, [1785].log_data[0].minminute := 15, [1785].log_data[0].maxminute := 15, [1785].log_data[0].valid := 1, [1785].log_data[1].valid := 1, [1785].log_data[2].valid := 1, [1785].log_data[3].valid := 1, [1785].log_data[4].valid := 1, [1785].time.Year := 2022, [1785].time.Month := 4, [1785].time.Day := 30, [1785].time.Hour := 2, [1785].time.Minute := 19, [1785].time.Second := 59, [1785].time.DST_ON := 1, [1786].log_data[0].min := 1.0, [1786].log_data[0].max := 1.0, [1786].log_data[0].total := 300.0, [1786].log_data[0].time := 300.0, [1786].log_data[0].minminute := 20, [1786].log_data[0].maxminute := 20, [1786].log_data[0].valid := 1, [1786].log_data[1].valid := 1, [1786].log_data[2].valid := 1, [1786].log_data[3].valid := 1, [1786].log_data[4].valid := 1, [1786].time.Year := 2022, [1786].time.Month := 4, [1786].time.Day := 30, [1786].time.Hour := 2, [1786].time.Minute := 24, [1786].time.Second := 59, [1786].time.DST_ON := 1, [1787].log_data[0].min := 1.0, [1787].log_data[0].max := 1.0, [1787].log_data[0].total := 300.0, [1787].log_data[0].time := 300.0, [1787].log_data[0].minminute := 25, [1787].log_data[0].maxminute := 25, [1787].log_data[0].valid := 1, [1787].log_data[1].valid := 1, [1787].log_data[2].valid := 1, [1787].log_data[3].valid := 1, [1787].log_data[4].valid := 1,
        [1787].time.Year := 2022, [1787].time.Month := 4, [1787].time.Day := 30, [1787].time.Hour := 2, [1787].time.Minute := 29, [1787].time.Second := 59, [1787].time.DST_ON := 1, [1788].log_data[0].min := 1.0, [1788].log_data[0].max := 1.0, [1788].log_data[0].total := 300.0, [1788].log_data[0].time := 300.0, [1788].log_data[0].minminute := 30, [1788].log_data[0].maxminute := 30, [1788].log_data[0].valid := 1, [1788].log_data[1].valid := 1, [1788].log_data[2].valid := 1, [1788].log_data[3].valid := 1, [1788].log_data[4].valid := 1, [1788].time.Year := 2022, [1788].time.Month := 4, [1788].time.Day := 30, [1788].time.Hour := 2, [1788].time.Minute := 34, [1788].time.Second := 59, [1788].time.DST_ON := 1, [1789].log_data[0].min := 1.0, [1789].log_data[0].max := 1.0, [1789].log_data[0].total := 300.0, [1789].log_data[0].time := 300.0, [1789].log_data[0].minminute := 35, [1789].log_data[0].maxminute := 35, [1789].log_data[0].valid := 1, [1789].log_data[1].valid := 1, [1789].log_data[2].valid := 1, [1789].log_data[3].valid := 1, [1789].log_data[4].valid := 1, [1789].time.Year := 2022, [1789].time.Month := 4, [1789].time.Day := 30, [1789].time.Hour := 2, [1789].time.Minute := 39, [1789].time.Second := 59, [1789].time.DST_ON := 1, [1790].log_data[0].min := 1.0, [1790].log_data[0].max := 1.0, [1790].log_data[0].total := 300.0, [1790].log_data[0].time := 300.0, [1790].log_data[0].minminute := 40, [1790].log_data[0].maxminute := 40, [1790].log_data[0].valid := 1, [1790].log_data[1].valid := 1, [1790].log_data[2].valid := 1, [1790].log_data[3].valid := 1, [1790].log_data[4].valid := 1, [1790].time.Year := 2022, [1790].time.Month := 4, [1790].time.Day := 30, [1790].time.Hour := 2, [1790].time.Minute := 44, [1790].time.Second := 59,
        [1790].time.DST_ON := 1, [1791].log_data[0].min := 1.0, [1791].log_data[0].max := 1.0, [1791].log_data[0].total := 300.0, [1791].log_data[0].time := 300.0, [1791].log_data[0].minminute := 45, [1791].log_data[0].maxminute := 45, [1791].log_data[0].valid := 1, [1791].log_data[1].valid := 1, [1791].log_data[2].valid := 1, [1791].log_data[3].valid := 1, [1791].log_data[4].valid := 1, [1791].time.Year := 2022, [1791].time.Month := 4, [1791].time.Day := 30, [1791].time.Hour := 2, [1791].time.Minute := 49, [1791].time.Second := 59, [1791].time.DST_ON := 1, [1792].log_data[0].min := 1.0, [1792].log_data[0].max := 1.0, [1792].log_data[0].total := 300.0, [1792].log_data[0].time := 300.0, [1792].log_data[0].minminute := 50, [1792].log_data[0].maxminute := 50, [1792].log_data[0].valid := 1, [1792].log_data[1].valid := 1, [1792].log_data[2].valid := 1, [1792].log_data[3].valid := 1, [1792].log_data[4].valid := 1, [1792].time.Year := 2022, [1792].time.Month := 4, [1792].time.Day := 30, [1792].time.Hour := 2, [1792].time.Minute := 54, [1792].time.Second := 59, [1792].time.DST_ON := 1, [1793].log_data[0].min := 1.0, [1793].log_data[0].max := 1.0, [1793].log_data[0].total := 300.0, [1793].log_data[0].time := 300.0, [1793].log_data[0].minminute := 55, [1793].log_data[0].maxminute := 55, [1793].log_data[0].valid := 1, [1793].log_data[1].valid := 1, [1793].log_data[2].valid := 1, [1793].log_data[3].valid := 1, [1793].log_data[4].valid := 1, [1793].time.Year := 2022, [1793].time.Month := 4, [1793].time.Day := 30, [1793].time.Hour := 2, [1793].time.Minute := 59, [1793].time.Second := 59, [1793].time.DST_ON := 1, [1794].log_data[0].min := 1.0, [1794].log_data[0].max := 1.0, [1794].log_data[0].total := 300.0, [1794].log_data[0].time := 300.0, [1794].log_data[0].valid := 1,
        [1794].log_data[1].valid := 1, [1794].log_data[2].valid := 1, [1794].log_data[3].valid := 1, [1794].log_data[4].valid := 1, [1794].time.Year := 2022, [1794].time.Month := 4, [1794].time.Day := 30, [1794].time.Hour := 3, [1794].time.Minute := 4, [1794].time.Second := 59, [1794].time.DST_ON := 1, [1795].log_data[0].min := 1.0, [1795].log_data[0].max := 1.0, [1795].log_data[0].total := 300.0, [1795].log_data[0].time := 300.0, [1795].log_data[0].minminute := 5, [1795].log_data[0].maxminute := 5, [1795].log_data[0].valid := 1, [1795].log_data[1].valid := 1, [1795].log_data[2].valid := 1, [1795].log_data[3].valid := 1, [1795].log_data[4].valid := 1, [1795].time.Year := 2022, [1795].time.Month := 4, [1795].time.Day := 30, [1795].time.Hour := 3, [1795].time.Minute := 9, [1795].time.Second := 59, [1795].time.DST_ON := 1, [1796].log_data[0].min := 1.0, [1796].log_data[0].max := 1.0, [1796].log_data[0].total := 300.0, [1796].log_data[0].time := 300.0, [1796].log_data[0].minminute := 10, [1796].log_data[0].maxminute := 10, [1796].log_data[0].valid := 1, [1796].log_data[1].valid := 1, [1796].log_data[2].valid := 1, [1796].log_data[3].valid := 1, [1796].log_data[4].valid := 1, [1796].time.Year := 2022, [1796].time.Month := 4, [1796].time.Day := 30, [1796].time.Hour := 3, [1796].time.Minute := 14, [1796].time.Second := 59, [1796].time.DST_ON := 1, [1797].log_data[0].min := 1.0, [1797].log_data[0].max := 1.0, [1797].log_data[0].total := 300.0, [1797].log_data[0].time := 300.0, [1797].log_data[0].minminute := 15, [1797].log_data[0].maxminute := 15, [1797].log_data[0].valid := 1, [1797].log_data[1].valid := 1, [1797].log_data[2].valid := 1, [1797].log_data[3].valid := 1, [1797].log_data[4].valid := 1, [1797].time.Year := 2022, [1797].time.Month := 4,
        [1797].time.Day := 30, [1797].time.Hour := 3, [1797].time.Minute := 19, [1797].time.Second := 59, [1797].time.DST_ON := 1, [1798].log_data[0].min := 1.0, [1798].log_data[0].max := 1.0, [1798].log_data[0].total := 300.0, [1798].log_data[0].time := 300.0, [1798].log_data[0].minminute := 20, [1798].log_data[0].maxminute := 20, [1798].log_data[0].valid := 1, [1798].log_data[1].valid := 1, [1798].log_data[2].valid := 1, [1798].log_data[3].valid := 1, [1798].log_data[4].valid := 1, [1798].time.Year := 2022, [1798].time.Month := 4, [1798].time.Day := 30, [1798].time.Hour := 3, [1798].time.Minute := 24, [1798].time.Second := 59, [1798].time.DST_ON := 1, [1799].log_data[0].min := 1.0, [1799].log_data[0].max := 1.0, [1799].log_data[0].total := 300.0, [1799].log_data[0].time := 300.0, [1799].log_data[0].minminute := 25, [1799].log_data[0].maxminute := 25, [1799].log_data[0].valid := 1, [1799].log_data[1].valid := 1, [1799].log_data[2].valid := 1, [1799].log_data[3].valid := 1, [1799].log_data[4].valid := 1, [1799].time.Year := 2022, [1799].time.Month := 4, [1799].time.Day := 30, [1799].time.Hour := 3, [1799].time.Minute := 29, [1799].time.Second := 59, [1799].time.DST_ON := 1, [1800].log_data[0].min := 1.0, [1800].log_data[0].max := 1.0, [1800].log_data[0].total := 300.0, [1800].log_data[0].time := 300.0, [1800].log_data[0].minminute := 30, [1800].log_data[0].maxminute := 30, [1800].log_data[0].valid := 1, [1800].log_data[1].valid := 1, [1800].log_data[2].valid := 1, [1800].log_data[3].valid := 1, [1800].log_data[4].valid := 1, [1800].time.Year := 2022, [1800].time.Month := 4, [1800].time.Day := 30, [1800].time.Hour := 3, [1800].time.Minute := 34, [1800].time.Second := 59, [1800].time.DST_ON := 1, [1801].log_data[0].min := 1.0,
        [1801].log_data[0].max := 1.0, [1801].log_data[0].total := 300.0, [1801].log_data[0].time := 300.0, [1801].log_data[0].minminute := 35, [1801].log_data[0].maxminute := 35, [1801].log_data[0].valid := 1, [1801].log_data[1].valid := 1, [1801].log_data[2].valid := 1, [1801].log_data[3].valid := 1, [1801].log_data[4].valid := 1, [1801].time.Year := 2022, [1801].time.Month := 4, [1801].time.Day := 30, [1801].time.Hour := 3, [1801].time.Minute := 39, [1801].time.Second := 59, [1801].time.DST_ON := 1, [1802].log_data[0].min := 1.0, [1802].log_data[0].max := 1.0, [1802].log_data[0].total := 300.0, [1802].log_data[0].time := 300.0, [1802].log_data[0].minminute := 40, [1802].log_data[0].maxminute := 40, [1802].log_data[0].valid := 1, [1802].log_data[1].valid := 1, [1802].log_data[2].valid := 1, [1802].log_data[3].valid := 1, [1802].log_data[4].valid := 1, [1802].time.Year := 2022, [1802].time.Month := 4, [1802].time.Day := 30, [1802].time.Hour := 3, [1802].time.Minute := 44, [1802].time.Second := 59, [1802].time.DST_ON := 1, [1803].log_data[0].min := 1.0, [1803].log_data[0].max := 1.0, [1803].log_data[0].total := 300.0, [1803].log_data[0].time := 300.0, [1803].log_data[0].minminute := 45, [1803].log_data[0].maxminute := 45, [1803].log_data[0].valid := 1, [1803].log_data[1].valid := 1, [1803].log_data[2].valid := 1, [1803].log_data[3].valid := 1, [1803].log_data[4].valid := 1, [1803].time.Year := 2022, [1803].time.Month := 4, [1803].time.Day := 30, [1803].time.Hour := 3, [1803].time.Minute := 49, [1803].time.Second := 59, [1803].time.DST_ON := 1, [1804].log_data[0].min := 1.0, [1804].log_data[0].max := 1.0, [1804].log_data[0].total := 300.0, [1804].log_data[0].time := 300.0, [1804].log_data[0].minminute := 50, [1804].log_data[0].maxminute := 50, [1804].log_data[0].valid := 1,
        [1804].log_data[1].valid := 1, [1804].log_data[2].valid := 1, [1804].log_data[3].valid := 1, [1804].log_data[4].valid := 1, [1804].time.Year := 2022, [1804].time.Month := 4, [1804].time.Day := 30, [1804].time.Hour := 3, [1804].time.Minute := 54, [1804].time.Second := 59, [1804].time.DST_ON := 1, [1805].log_data[0].min := 1.0, [1805].log_data[0].max := 1.0, [1805].log_data[0].total := 300.0, [1805].log_data[0].time := 300.0, [1805].log_data[0].minminute := 55, [1805].log_data[0].maxminute := 55, [1805].log_data[0].valid := 1, [1805].log_data[1].valid := 1, [1805].log_data[2].valid := 1, [1805].log_data[3].valid := 1, [1805].log_data[4].valid := 1, [1805].time.Year := 2022, [1805].time.Month := 4, [1805].time.Day := 30, [1805].time.Hour := 3, [1805].time.Minute := 59, [1805].time.Second := 59, [1805].time.DST_ON := 1, [1806].log_data[0].min := 1.0, [1806].log_data[0].max := 1.0, [1806].log_data[0].total := 300.0, [1806].log_data[0].time := 300.0, [1806].log_data[0].valid := 1, [1806].log_data[1].valid := 1, [1806].log_data[2].valid := 1, [1806].log_data[3].valid := 1, [1806].log_data[4].valid := 1, [1806].time.Year := 2022, [1806].time.Month := 4, [1806].time.Day := 30, [1806].time.Hour := 4, [1806].time.Minute := 4, [1806].time.Second := 59, [1806].time.DST_ON := 1, [1807].log_data[0].min := 1.0, [1807].log_data[0].max := 1.0, [1807].log_data[0].total := 300.0, [1807].log_data[0].time := 300.0, [1807].log_data[0].minminute := 5, [1807].log_data[0].maxminute := 5, [1807].log_data[0].valid := 1, [1807].log_data[1].valid := 1, [1807].log_data[2].valid := 1, [1807].log_data[3].valid := 1, [1807].log_data[4].valid := 1, [1807].time.Year := 2022, [1807].time.Month := 4, [1807].time.Day := 30, [1807].time.Hour := 4,
